LIN {X 0,Y 476.496,Z 164.694,A -85,B 0,C 180,E1 -7312.32,E2 -7312.32} C_VEL
LIN {X 0,Y 474.632,Z 154.455,A -85,B 0,C 180,E1 -7314.435,E2 -7314.435} C_VEL
LIN {X 0,Y 474.635,Z 154.349,A -85,B 0,C 180,E1 -7317.323,E2 -7317.323} C_VEL
LIN {X 0,Y 474.598,Z 154.362,A -85,B 0,C 180,E1 -7320.229,E2 -7320.229} C_VEL
LIN {X 0,Y 474.631,Z 154.36,A -85,B 0,C 180,E1 -7323.22,E2 -7323.22} C_VEL
LIN {X 0,Y 474.579,Z 154.367,A -85,B 0,C 180,E1 -7326.323,E2 -7326.323} C_VEL
LIN {X 0,Y 474.62,Z 154.363,A -85,B 0,C 180,E1 -7329.547,E2 -7329.547} C_VEL
LIN {X 0,Y 474.593,Z 154.363,A -85,B 0,C 180,E1 -7332.232,E2 -7332.232} C_VEL
LIN {X 0,Y 474.614,Z 154.365,A -85,B 0,C 180,E1 -7335.296,E2 -7335.296} C_VEL
LIN {X 0,Y 474.612,Z 154.36,A -85,B 0,C 180,E1 -7338.214,E2 -7338.214} C_VEL
LIN {X 0,Y 474.602,Z 154.355,A -85,B 0,C 180,E1 -7341.542,E2 -7341.542} C_VEL
LIN {X 0,Y 474.614,Z 154.352,A -85,B 0,C 180,E1 -7344.725,E2 -7344.725} C_VEL
LIN {X 0,Y 474.624,Z 154.36,A -85,B 0,C 180,E1 -7347.787,E2 -7347.787} C_VEL
LIN {X 0,Y 474.611,Z 154.363,A -85,B 0,C 180,E1 -7350.884,E2 -7350.884} C_VEL
LIN {X 0,Y 474.642,Z 154.358,A -85,B 0,C 180,E1 -7353.627,E2 -7353.627} C_VEL
LIN {X 0,Y 474.623,Z 154.359,A -85,B 0,C 180,E1 -7356.641,E2 -7356.641} C_VEL
LIN {X 0,Y 474.642,Z 154.358,A -85,B 0,C 180,E1 -7360.089,E2 -7360.089} C_VEL
LIN {X 0,Y 474.626,Z 154.36,A -85,B 0,C 180,E1 -7362.774,E2 -7362.774} C_VEL
LIN {X 0,Y 474.634,Z 154.359,A -85,B 0,C 180,E1 -7365.421,E2 -7365.421} C_VEL
LIN {X 0,Y 474.728,Z 154.343,A -85,B 0,C 180,E1 -7368.038,E2 -7368.038} C_VEL
LIN {X 0,Y 474.714,Z 154.348,A -85,B 0,C 180,E1 -7371.486,E2 -7371.486} C_VEL
LIN {X 0,Y 474.756,Z 154.343,A -85,B 0,C 180,E1 -7374.052,E2 -7374.052} C_VEL
LIN {X 0,Y 474.879,Z 154.327,A -85,B 0,C 180,E1 -7377.455,E2 -7377.455} C_VEL
LIN {X 0,Y 474.844,Z 154.331,A -85,B 0,C 180,E1 -7380.848,E2 -7380.848} C_VEL
LIN {X 0,Y 474.879,Z 154.327,A -85,B 0,C 180,E1 -7382.545,E2 -7382.545} C_VEL
LIN {X 0,Y 474.756,Z 154.345,A -85,B 0,C 180,E1 -7385.948,E2 -7385.948} C_VEL
LIN {X 0,Y 474.715,Z 154.346,A -85,B 0,C 180,E1 -7388.514,E2 -7388.514} C_VEL
LIN {X 0,Y 474.692,Z 154.353,A -85,B 0,C 180,E1 -7391.963,E2 -7391.963} C_VEL
LIN {X 0,Y 474.687,Z 154.346,A -85,B 0,C 180,E1 -7395.456,E2 -7395.456} C_VEL
LIN {X 0,Y 474.654,Z 154.356,A -85,B 0,C 180,E1 -7399.011,E2 -7399.011} C_VEL
LIN {X 0,Y 474.582,Z 154.363,A -85,B 0,C 180,E1 -7401.729,E2 -7401.729} C_VEL
LIN {X 0,Y 474.648,Z 154.361,A -85,B 0,C 180,E1 -7404.494,E2 -7404.494} C_VEL
LIN {X 0,Y 474.671,Z 154.35,A -85,B 0,C 180,E1 -7407.335,E2 -7407.335} C_VEL
LIN {X 0,Y 474.595,Z 154.37,A -85,B 0,C 180,E1 -7410.231,E2 -7410.231} C_VEL
LIN {X 0,Y 474.633,Z 154.352,A -85,B 0,C 180,E1 -7413.221,E2 -7413.221} C_VEL
LIN {X 0,Y 474.583,Z 154.357,A -85,B 0,C 180,E1 -7416.324,E2 -7416.324} C_VEL
LIN {X 0,Y 474.619,Z 154.364,A -85,B 0,C 180,E1 -7419.649,E2 -7419.649} C_VEL
LIN {X 0,Y 474.599,Z 154.351,A -85,B 0,C 180,E1 -7422.936,E2 -7422.936} C_VEL
LIN {X 0,Y 474.598,Z 154.367,A -85,B 0,C 180,E1 -7425.896,E2 -7425.896} C_VEL
LIN {X 0,Y 474.622,Z 154.355,A -85,B 0,C 180,E1 -7429.042,E2 -7429.042} C_VEL
LIN {X 0,Y 474.605,Z 154.362,A -85,B 0,C 180,E1 -7431.705,E2 -7431.705} C_VEL
LIN {X 0,Y 474.624,Z 154.355,A -85,B 0,C 180,E1 -7434.727,E2 -7434.727} C_VEL
LIN {X 0,Y 474.633,Z 154.363,A -85,B 0,C 180,E1 -7437.789,E2 -7437.789} C_VEL
LIN {X 0,Y 474.621,Z 154.362,A -85,B 0,C 180,E1 -7440.886,E2 -7440.886} C_VEL
LIN {X 0,Y 474.657,Z 154.36,A -85,B 0,C 180,E1 -7443.629,E2 -7443.629} C_VEL
LIN {X 0,Y 474.661,Z 154.46,A -85,B 0,C 180,E1 -7446.902,E2 -7446.902} C_VEL
LIN {X 0,Y 476.247,Z 163.612,A -85,B 0,C 180,E1 -7448.865,E2 -7448.865} C_VEL
LIN {X 0,Y 476.003,Z 169.231,A -85,B 0,C 180,E1 -7449.97,E2 -7449.97} C_VEL
LIN {X 0,Y 475.26,Z 171.385,A -85,B 0,C 180,E1 -7450.363,E2 -7450.363} C_VEL
LIN {X 0,Y 472.299,Z 175.015,A -85,B 0,C 180,E1 -7450.95,E2 -7450.95} C_VEL
LIN {X 0,Y 469.331,Z 178.656,A -85,B 0,C 180,E1 -7451.543,E2 -7451.543} C_VEL
LIN {X 0,Y 468.592,Z 180.83,A -85,B 0,C 180,E1 -7451.942,E2 -7451.942} C_VEL
LIN {X 0,Y 468.452,Z 186.605,A -85,B 0,C 180,E1 -7453.017,E2 -7453.017} C_VEL
LIN {X 0,Y 471.25,Z 202.144,A -85,B 0,C 180,E1 -7453.391,E2 -7453.391} C_VEL
LIN {X 0,Y 470.685,Z 294.202,A -85,B 0,C 180,E1 -7454.826,E2 -7454.826} C_VEL
LIN {X 0,Y 470.344,Z 307.324,A -85,B 0,C 180,E1 -7455.202,E2 -7455.202} C_VEL
LIN {X 0,Y 469.901,Z 319.4,A -85,B 0,C 180,E1 -7455.714,E2 -7455.714} C_VEL
LIN {X 0,Y 469.477,Z 330.795,A -85,B 0,C 180,E1 -7456.364,E2 -7456.364} C_VEL
LIN {X 0,Y 469.045,Z 342.481,A -85,B 0,C 180,E1 -7457.232,E2 -7457.232} C_VEL
LIN {X 0,Y 468.521,Z 352.971,A -85,B 0,C 180,E1 -7458.207,E2 -7458.207} C_VEL
LIN {X 0,Y 468.048,Z 361.544,A -85,B 0,C 180,E1 -7459.182,E2 -7459.182} C_VEL
LIN {X 0,Y 467.675,Z 369.442,A -85,B 0,C 180,E1 -7460.267,E2 -7460.267} C_VEL
LIN {X 0,Y 467.268,Z 377.166,A -85,B 0,C 180,E1 -7461.568,E2 -7461.568} C_VEL
LIN {X 0,Y 466.994,Z 384.254,A -85,B 0,C 180,E1 -7463.086,E2 -7463.086} C_VEL
LIN {X 0,Y 466.881,Z 388.978,A -85,B 0,C 180,E1 -7464.385,E2 -7464.385} C_VEL
LIN {X 0,Y 466.691,Z 392.597,A -85,B 0,C 180,E1 -7465.682,E2 -7465.682} C_VEL
LIN {X 0,Y 466.746,Z 394.466,A -85,B 0,C 180,E1 -7466.547,E2 -7466.547} C_VEL
LIN {X 0,Y 466.669,Z 395.877,A -85,B 0,C 180,E1 -7467.411,E2 -7467.411} C_VEL
LIN {X 0,Y 466.59,Z 397.498,A -85,B 0,C 180,E1 -7469.137,E2 -7469.137} C_VEL
LIN {X 0,Y 466.599,Z 397.734,A -85,B 0,C 180,E1 -7470,E2 -7470} C_VEL
LIN {X 0,Y 466.59,Z 397.547,A -85,B 0,C 180,E1 -7470.863,E2 -7470.863} C_VEL
LIN {X 0,Y 466.669,Z 395.992,A -85,B 0,C 180,E1 -7472.59,E2 -7472.59} C_VEL
LIN {X 0,Y 466.745,Z 394.631,A -85,B 0,C 180,E1 -7473.453,E2 -7473.453} C_VEL
LIN {X 0,Y 466.712,Z 391.756,A -85,B 0,C 180,E1 -7474.751,E2 -7474.751} C_VEL
LIN {X 0,Y 466.89,Z 387.046,A -85,B 0,C 180,E1 -7476.28,E2 -7476.28} C_VEL
LIN {X 0,Y 467.102,Z 380.85,A -85,B 0,C 180,E1 -7477.783,E2 -7477.783} C_VEL
LIN {X 0,Y 467.471,Z 374.044,A -85,B 0,C 180,E1 -7479.083,E2 -7479.083} C_VEL
LIN {X 0,Y 467.839,Z 365.548,A -85,B 0,C 180,E1 -7480.385,E2 -7480.385} C_VEL
LIN {X 0,Y 468.279,Z 356.811,A -85,B 0,C 180,E1 -7481.47,E2 -7481.47} C_VEL
LIN {X 0,Y 468.838,Z 346.297,A -85,B 0,C 180,E1 -7482.531,E2 -7482.531} C_VEL
LIN {X 0,Y 469.248,Z 335.279,A -85,B 0,C 180,E1 -7483.423,E2 -7483.423} C_VEL
LIN {X 0,Y 469.803,Z 323.169,A -85,B 0,C 180,E1 -7484.18,E2 -7484.18} C_VEL
LIN {X 0,Y 470.239,Z 310.502,A -85,B 0,C 180,E1 -7484.774,E2 -7484.774} C_VEL
LIN {X 0,Y 470.602,Z 297.977,A -85,B 0,C 180,E1 -7485.178,E2 -7485.178} C_VEL
LIN {X 0,Y 470.757,Z 281.99,A -85,B 0,C 180,E1 -7485.477,E2 -7485.477} C_VEL
LIN {X 0,Y 471.183,Z 201.775,A -85,B 0,C 180,E1 -7486.71,E2 -7486.71} C_VEL
LIN {X 0,Y 468.503,Z 186.823,A -85,B 0,C 180,E1 -7487.063,E2 -7487.063} C_VEL
LIN {X 0,Y 468.44,Z 185.986,A -85,B 0,C 180,E1 -7487.157,E2 -7487.157} C_VEL
LIN {X 0,Y 469.081,Z 169.504,A -85,B 0,C 180,E1 -7490.386,E2 -7490.386} C_VEL
LIN {X 0,Y 469.266,Z 164.503,A -85,B 0,C 180,E1 -7491.386,E2 -7491.386} C_VEL
LIN {X 0,Y 467.613,Z 155.303,A -85,B 0,C 180,E1 -7493.404,E2 -7493.404} C_VEL
LIN {X 0,Y 467.618,Z 155.238,A -85,B 0,C 180,E1 -7496.8,E2 -7496.8} C_VEL
LIN {X 0,Y 467.555,Z 155.243,A -85,B 0,C 180,E1 -7499.738,E2 -7499.738} C_VEL
LIN {X 0,Y 467.584,Z 155.241,A -85,B 0,C 180,E1 -7502.758,E2 -7502.758} C_VEL
LIN {X 0,Y 467.556,Z 155.238,A -85,B 0,C 180,E1 -7505.889,E2 -7505.889} C_VEL
LIN {X 0,Y 467.559,Z 155.234,A -85,B 0,C 180,E1 -7509.146,E2 -7509.146} C_VEL
LIN {X 0,Y 467.585,Z 155.24,A -85,B 0,C 180,E1 -7512.566,E2 -7512.566} C_VEL
LIN {X 0,Y 467.563,Z 155.235,A -85,B 0,C 180,E1 -7515.052,E2 -7515.052} C_VEL
LIN {X 0,Y 467.587,Z 155.225,A -85,B 0,C 180,E1 -7517.439,E2 -7517.439} C_VEL
LIN {X 0,Y 467.579,Z 155.238,A -85,B 0,C 180,E1 -7520.855,E2 -7520.855} C_VEL
LIN {X 0,Y 467.558,Z 155.223,A -85,B 0,C 180,E1 -7524.26,E2 -7524.26} C_VEL
LIN {X 0,Y 467.577,Z 155.232,A -85,B 0,C 180,E1 -7527.32,E2 -7527.32} C_VEL
LIN {X 0,Y 467.565,Z 155.239,A -85,B 0,C 180,E1 -7530.667,E2 -7530.667} C_VEL
LIN {X 0,Y 467.607,Z 155.23,A -85,B 0,C 180,E1 -7533.199,E2 -7533.199} C_VEL
LIN {X 0,Y 467.584,Z 155.235,A -85,B 0,C 180,E1 -7536.469,E2 -7536.469} C_VEL
LIN {X 0,Y 467.616,Z 155.237,A -85,B 0,C 180,E1 -7539.777,E2 -7539.777} C_VEL
LIN {X 0,Y 467.6,Z 155.233,A -85,B 0,C 180,E1 -7542.506,E2 -7542.506} C_VEL
LIN {X 0,Y 467.599,Z 155.23,A -85,B 0,C 180,E1 -7545.196,E2 -7545.196} C_VEL
LIN {X 0,Y 467.649,Z 155.233,A -85,B 0,C 180,E1 -7547.854,E2 -7547.854} C_VEL
LIN {X 0,Y 467.674,Z 155.221,A -85,B 0,C 180,E1 -7551.357,E2 -7551.357} C_VEL
LIN {X 0,Y 467.726,Z 155.222,A -85,B 0,C 180,E1 -7553.962,E2 -7553.962} C_VEL
LIN {X 0,Y 467.849,Z 155.202,A -85,B 0,C 180,E1 -7557.417,E2 -7557.417} C_VEL
LIN {X 0,Y 467.872,Z 155.203,A -85,B 0,C 180,E1 -7560,E2 -7560} C_VEL
LIN {X 0,Y 467.85,Z 155.202,A -85,B 0,C 180,E1 -7562.583,E2 -7562.583} C_VEL
LIN {X 0,Y 467.725,Z 155.218,A -85,B 0,C 180,E1 -7566.038,E2 -7566.038} C_VEL
LIN {X 0,Y 467.662,Z 155.227,A -85,B 0,C 180,E1 -7568.643,E2 -7568.643} C_VEL
LIN {X 0,Y 467.648,Z 155.225,A -85,B 0,C 180,E1 -7572.146,E2 -7572.146} C_VEL
LIN {X 0,Y 467.632,Z 155.232,A -85,B 0,C 180,E1 -7575.695,E2 -7575.695} C_VEL
LIN {X 0,Y 467.615,Z 155.236,A -85,B 0,C 180,E1 -7579.308,E2 -7579.308} C_VEL
LIN {X 0,Y 467.527,Z 155.243,A -85,B 0,C 180,E1 -7582.074,E2 -7582.074} C_VEL
LIN {X 0,Y 467.578,Z 155.236,A -85,B 0,C 180,E1 -7584.889,E2 -7584.889} C_VEL
LIN {X 0,Y 467.613,Z 155.233,A -85,B 0,C 180,E1 -7587.77,E2 -7587.77} C_VEL
LIN {X 0,Y 467.562,Z 155.244,A -85,B 0,C 180,E1 -7591.045,E2 -7591.045} C_VEL
LIN {X 0,Y 467.572,Z 155.235,A -85,B 0,C 180,E1 -7594.241,E2 -7594.241} C_VEL
LIN {X 0,Y 467.543,Z 155.231,A -85,B 0,C 180,E1 -7597.187,E2 -7597.187} C_VEL
LIN {X 0,Y 467.567,Z 155.239,A -85,B 0,C 180,E1 -7600.266,E2 -7600.266} C_VEL
LIN {X 0,Y 467.545,Z 155.241,A -85,B 0,C 180,E1 -7603.746,E2 -7603.746} C_VEL
LIN {X 0,Y 467.544,Z 155.243,A -85,B 0,C 180,E1 -7606.255,E2 -7606.255} C_VEL
LIN {X 0,Y 467.557,Z 155.239,A -85,B 0,C 180,E1 -7609.734,E2 -7609.734} C_VEL
LIN {X 0,Y 467.541,Z 155.242,A -85,B 0,C 180,E1 -7612.815,E2 -7612.815} C_VEL
LIN {X 0,Y 467.583,Z 155.234,A -85,B 0,C 180,E1 -7616.212,E2 -7616.212} C_VEL
LIN {X 0,Y 467.567,Z 155.238,A -85,B 0,C 180,E1 -7619.266,E2 -7619.266} C_VEL
LIN {X 0,Y 467.604,Z 155.225,A -85,B 0,C 180,E1 -7622.469,E2 -7622.469} C_VEL
LIN {X 0,Y 467.608,Z 155.32,A -85,B 0,C 180,E1 -7625.35,E2 -7625.35} C_VEL
LIN {X 0,Y 469.554,Z 165.837,A -85,B 0,C 180,E1 -7627.563,E2 -7627.563} C_VEL
LIN {X 0,Y 469.08,Z 177.76,A -85,B 0,C 180,E1 -7629.843,E2 -7629.843} C_VEL
LIN {X 0,Y 468.446,Z 192.056,A -85,B 0,C 180,E1 -7632.539,E2 -7632.539} C_VEL
LIN {X 0,Y 468.409,Z 194.559,A -85,B 0,C 180,E1 -7632.963,E2 -7632.963} C_VEL
LIN {X 0,Y 471.306,Z 212.054,A -85,B 0,C 180,E1 -7633.371,E2 -7633.371} C_VEL
LIN {X 0,Y 470.62,Z 302.152,A -85,B 0,C 180,E1 -7634.768,E2 -7634.768} C_VEL
LIN {X 0,Y 470.222,Z 315.409,A -85,B 0,C 180,E1 -7635.142,E2 -7635.142} C_VEL
LIN {X 0,Y 469.849,Z 327.558,A -85,B 0,C 180,E1 -7635.656,E2 -7635.656} C_VEL
LIN {X 0,Y 469.374,Z 339.815,A -85,B 0,C 180,E1 -7636.36,E2 -7636.36} C_VEL
LIN {X 0,Y 468.891,Z 350.559,A -85,B 0,C 180,E1 -7637.157,E2 -7637.157} C_VEL
LIN {X 0,Y 468.41,Z 361.811,A -85,B 0,C 180,E1 -7638.204,E2 -7638.204} C_VEL
LIN {X 0,Y 467.898,Z 370.327,A -85,B 0,C 180,E1 -7639.178,E2 -7639.178} C_VEL
LIN {X 0,Y 467.514,Z 378.184,A -85,B 0,C 180,E1 -7640.263,E2 -7640.263} C_VEL
LIN {X 0,Y 467.179,Z 385.855,A -85,B 0,C 180,E1 -7641.566,E2 -7641.566} C_VEL
LIN {X 0,Y 466.855,Z 392.925,A -85,B 0,C 180,E1 -7643.083,E2 -7643.083} C_VEL
LIN {X 0,Y 466.801,Z 397.628,A -85,B 0,C 180,E1 -7644.384,E2 -7644.384} C_VEL
LIN {X 0,Y 466.648,Z 401.219,A -85,B 0,C 180,E1 -7645.681,E2 -7645.681} C_VEL
LIN {X 0,Y 466.69,Z 403.072,A -85,B 0,C 180,E1 -7646.546,E2 -7646.546} C_VEL
LIN {X 0,Y 466.646,Z 404.461,A -85,B 0,C 180,E1 -7647.41,E2 -7647.41} C_VEL
LIN {X 0,Y 466.589,Z 406.056,A -85,B 0,C 180,E1 -7649.137,E2 -7649.137} C_VEL
LIN {X 0,Y 466.598,Z 406.272,A -85,B 0,C 180,E1 -7650,E2 -7650} C_VEL
LIN {X 0,Y 466.604,Z 405.452,A -85,B 0,C 180,E1 -7651.726,E2 -7651.726} C_VEL
LIN {X 0,Y 466.646,Z 404.463,A -85,B 0,C 180,E1 -7652.589,E2 -7652.589} C_VEL
LIN {X 0,Y 466.689,Z 403.074,A -85,B 0,C 180,E1 -7653.453,E2 -7653.453} C_VEL
LIN {X 0,Y 466.692,Z 400.152,A -85,B 0,C 180,E1 -7654.751,E2 -7654.751} C_VEL
LIN {X 0,Y 466.8,Z 396.197,A -85,B 0,C 180,E1 -7656.049,E2 -7656.049} C_VEL
LIN {X 0,Y 466.988,Z 390.112,A -85,B 0,C 180,E1 -7657.566,E2 -7657.566} C_VEL
LIN {X 0,Y 467.303,Z 383.46,A -85,B 0,C 180,E1 -7658.867,E2 -7658.867} C_VEL
LIN {X 0,Y 467.693,Z 375.204,A -85,B 0,C 180,E1 -7660.169,E2 -7660.169} C_VEL
LIN {X 0,Y 468.102,Z 366.74,A -85,B 0,C 180,E1 -7661.255,E2 -7661.255} C_VEL
LIN {X 0,Y 468.662,Z 356.491,A -85,B 0,C 180,E1 -7662.318,E2 -7662.318} C_VEL
LIN {X 0,Y 469.058,Z 346.211,A -85,B 0,C 180,E1 -7663.185,E2 -7663.185} C_VEL
LIN {X 0,Y 469.515,Z 334.567,A -85,B 0,C 180,E1 -7663.967,E2 -7663.967} C_VEL
LIN {X 0,Y 469.994,Z 322.917,A -85,B 0,C 180,E1 -7664.56,E2 -7664.56} C_VEL
LIN {X 0,Y 470.42,Z 309.487,A -85,B 0,C 180,E1 -7665.044,E2 -7665.044} C_VEL
LIN {X 0,Y 470.693,Z 296.212,A -85,B 0,C 180,E1 -7665.34,E2 -7665.34} C_VEL
LIN {X 0,Y 471.296,Z 211.905,A -85,B 0,C 180,E1 -7666.629,E2 -7666.629} C_VEL
LIN {X 0,Y 468.42,Z 194.62,A -85,B 0,C 180,E1 -7667.029,E2 -7667.029} C_VEL
LIN {X 0,Y 468.91,Z 181.321,A -85,B 0,C 180,E1 -7669.479,E2 -7669.479} C_VEL
LIN {X 0,Y 469.584,Z 167.014,A -85,B 0,C 180,E1 -7672.203,E2 -7672.203} C_VEL
LIN {X 0,Y 468.738,Z 161.245,A -85,B 0,C 180,E1 -7673.37,E2 -7673.37} C_VEL
LIN {X 0,Y 467.606,Z 155.311,A -85,B 0,C 180,E1 -7674.649,E2 -7674.649} C_VEL
LIN {X 0,Y 467.578,Z 155.231,A -85,B 0,C 180,E1 -7677.771,E2 -7677.771} C_VEL
LIN {X 0,Y 467.564,Z 155.24,A -85,B 0,C 180,E1 -7681.044,E2 -7681.044} C_VEL
LIN {X 0,Y 467.584,Z 155.233,A -85,B 0,C 180,E1 -7684.241,E2 -7684.241} C_VEL
LIN {X 0,Y 467.538,Z 155.242,A -85,B 0,C 180,E1 -7687.184,E2 -7687.184} C_VEL
LIN {X 0,Y 467.564,Z 155.238,A -85,B 0,C 180,E1 -7690.264,E2 -7690.264} C_VEL
LIN {X 0,Y 467.544,Z 155.243,A -85,B 0,C 180,E1 -7693.744,E2 -7693.744} C_VEL
LIN {X 0,Y 467.549,Z 155.24,A -85,B 0,C 180,E1 -7696.255,E2 -7696.255} C_VEL
LIN {X 0,Y 467.57,Z 155.242,A -85,B 0,C 180,E1 -7698.722,E2 -7698.722} C_VEL
LIN {X 0,Y 467.556,Z 155.231,A -85,B 0,C 180,E1 -7701.954,E2 -7701.954} C_VEL
LIN {X 0,Y 467.554,Z 155.238,A -85,B 0,C 180,E1 -7705.166,E2 -7705.166} C_VEL
LIN {X 0,Y 467.571,Z 155.24,A -85,B 0,C 180,E1 -7708.259,E2 -7708.259} C_VEL
LIN {X 0,Y 467.564,Z 155.241,A -85,B 0,C 180,E1 -7711.249,E2 -7711.249} C_VEL
LIN {X 0,Y 467.585,Z 155.237,A -85,B 0,C 180,E1 -7714.159,E2 -7714.159} C_VEL
LIN {X 0,Y 467.564,Z 155.243,A -85,B 0,C 180,E1 -7716.995,E2 -7716.995} C_VEL
LIN {X 0,Y 467.61,Z 155.233,A -85,B 0,C 180,E1 -7719.777,E2 -7719.777} C_VEL
LIN {X 0,Y 467.586,Z 155.234,A -85,B 0,C 180,E1 -7722.506,E2 -7722.506} C_VEL
LIN {X 0,Y 467.592,Z 155.238,A -85,B 0,C 180,E1 -7725.196,E2 -7725.196} C_VEL
LIN {X 0,Y 467.671,Z 155.221,A -85,B 0,C 180,E1 -7727.855,E2 -7727.855} C_VEL
LIN {X 0,Y 467.668,Z 155.227,A -85,B 0,C 180,E1 -7731.357,E2 -7731.357} C_VEL
LIN {X 0,Y 467.72,Z 155.218,A -85,B 0,C 180,E1 -7733.962,E2 -7733.962} C_VEL
LIN {X 0,Y 467.845,Z 155.203,A -85,B 0,C 180,E1 -7737.417,E2 -7737.417} C_VEL
LIN {X 0,Y 467.867,Z 155.203,A -85,B 0,C 180,E1 -7740,E2 -7740} C_VEL
LIN {X 0,Y 467.845,Z 155.203,A -85,B 0,C 180,E1 -7742.583,E2 -7742.583} C_VEL
LIN {X 0,Y 467.721,Z 155.222,A -85,B 0,C 180,E1 -7746.038,E2 -7746.038} C_VEL
LIN {X 0,Y 467.669,Z 155.222,A -85,B 0,C 180,E1 -7748.643,E2 -7748.643} C_VEL
LIN {X 0,Y 467.643,Z 155.233,A -85,B 0,C 180,E1 -7752.146,E2 -7752.146} C_VEL
LIN {X 0,Y 467.627,Z 155.226,A -85,B 0,C 180,E1 -7755.696,E2 -7755.696} C_VEL
LIN {X 0,Y 467.606,Z 155.236,A -85,B 0,C 180,E1 -7758.765,E2 -7758.765} C_VEL
LIN {X 0,Y 467.571,Z 155.234,A -85,B 0,C 180,E1 -7761.269,E2 -7761.269} C_VEL
LIN {X 0,Y 467.563,Z 155.241,A -85,B 0,C 180,E1 -7763.944,E2 -7763.944} C_VEL
LIN {X 0,Y 467.606,Z 155.231,A -85,B 0,C 180,E1 -7766.801,E2 -7766.801} C_VEL
LIN {X 0,Y 467.544,Z 155.243,A -85,B 0,C 180,E1 -7769.739,E2 -7769.739} C_VEL
LIN {X 0,Y 467.574,Z 155.232,A -85,B 0,C 180,E1 -7772.759,E2 -7772.759} C_VEL
LIN {X 0,Y 467.547,Z 155.226,A -85,B 0,C 180,E1 -7775.89,E2 -7775.89} C_VEL
LIN {X 0,Y 467.574,Z 155.238,A -85,B 0,C 180,E1 -7779.146,E2 -7779.146} C_VEL
LIN {X 0,Y 467.58,Z 155.227,A -85,B 0,C 180,E1 -7782.568,E2 -7782.568} C_VEL
LIN {X 0,Y 467.559,Z 155.235,A -85,B 0,C 180,E1 -7785.054,E2 -7785.054} C_VEL
LIN {X 0,Y 467.583,Z 155.24,A -85,B 0,C 180,E1 -7787.441,E2 -7787.441} C_VEL
LIN {X 0,Y 467.555,Z 155.234,A -85,B 0,C 180,E1 -7790.854,E2 -7790.854} C_VEL
LIN {X 0,Y 467.558,Z 155.237,A -85,B 0,C 180,E1 -7794.262,E2 -7794.262} C_VEL
LIN {X 0,Y 467.579,Z 155.241,A -85,B 0,C 180,E1 -7797.322,E2 -7797.322} C_VEL
LIN {X 0,Y 467.567,Z 155.241,A -85,B 0,C 180,E1 -7800.669,E2 -7800.669} C_VEL
LIN {X 0,Y 467.614,Z 155.238,A -85,B 0,C 180,E1 -7803.201,E2 -7803.201} C_VEL
LIN {X 0,Y 467.618,Z 155.252,A -85,B 0,C 180,E1 -7806.627,E2 -7806.627} C_VEL
LIN {X 0,Y 467.7,Z 155.798,A -85,B 0,C 180,E1 -7806.847,E2 -7806.847} C_VEL
LIN {X 0,Y 469.198,Z 164.087,A -85,B 0,C 180,E1 -7808.62,E2 -7808.62} C_VEL
LIN {X 0,Y 468.839,Z 175.747,A -85,B 0,C 180,E1 -7810.945,E2 -7810.945} C_VEL
LIN {X 0,Y 468.592,Z 180.83,A -85,B 0,C 180,E1 -7811.942,E2 -7811.942} C_VEL
LIN {X 0,Y 468.359,Z 183.305,A -85,B 0,C 180,E1 -7812.302,E2 -7812.302} C_VEL
LIN {X 0,Y 467.542,Z 188.103,A -85,B 0,C 180,E1 -7812.697,E2 -7812.697} C_VEL
LIN {X 0,Y 466.477,Z 193.563,A -85,B 0,C 180,E1 -7812.946,E2 -7812.946} C_VEL
LIN {X 0,Y 465.076,Z 201.654,A -85,B 0,C 180,E1 -7813.136,E2 -7813.136} C_VEL
LIN {X 0,Y 464.452,Z 209.922,A -85,B 0,C 180,E1 -7813.262,E2 -7813.262} C_VEL
LIN {X 0,Y 463.85,Z 294.285,A -85,B 0,C 180,E1 -7814.597,E2 -7814.597} C_VEL
LIN {X 0,Y 463.475,Z 307.401,A -85,B 0,C 180,E1 -7814.978,E2 -7814.978} C_VEL
LIN {X 0,Y 463.005,Z 320.582,A -85,B 0,C 180,E1 -7815.552,E2 -7815.552} C_VEL
LIN {X 0,Y 462.51,Z 332.459,A -85,B 0,C 180,E1 -7816.266,E2 -7816.266} C_VEL
LIN {X 0,Y 462.058,Z 343.922,A -85,B 0,C 180,E1 -7817.155,E2 -7817.155} C_VEL
LIN {X 0,Y 461.512,Z 354.103,A -85,B 0,C 180,E1 -7818.137,E2 -7818.137} C_VEL
LIN {X 0,Y 460.983,Z 363.314,A -85,B 0,C 180,E1 -7819.237,E2 -7819.237} C_VEL
LIN {X 0,Y 460.49,Z 372.258,A -85,B 0,C 180,E1 -7820.558,E2 -7820.558} C_VEL
LIN {X 0,Y 460.107,Z 379.461,A -85,B 0,C 180,E1 -7821.878,E2 -7821.878} C_VEL
LIN {X 0,Y 459.895,Z 385.855,A -85,B 0,C 180,E1 -7823.373,E2 -7823.373} C_VEL
LIN {X 0,Y 459.738,Z 390.365,A -85,B 0,C 180,E1 -7824.738,E2 -7824.738} C_VEL
LIN {X 0,Y 459.604,Z 392.663,A -85,B 0,C 180,E1 -7825.616,E2 -7825.616} C_VEL
LIN {X 0,Y 459.643,Z 394.532,A -85,B 0,C 180,E1 -7826.494,E2 -7826.494} C_VEL
LIN {X 0,Y 459.593,Z 395.942,A -85,B 0,C 180,E1 -7827.371,E2 -7827.371} C_VEL
LIN {X 0,Y 459.495,Z 397.563,A -85,B 0,C 180,E1 -7829.124,E2 -7829.124} C_VEL
LIN {X 0,Y 459.501,Z 397.799,A -85,B 0,C 180,E1 -7830,E2 -7830} C_VEL
LIN {X 0,Y 459.495,Z 397.612,A -85,B 0,C 180,E1 -7830.877,E2 -7830.877} C_VEL
LIN {X 0,Y 459.593,Z 396.056,A -85,B 0,C 180,E1 -7832.63,E2 -7832.63} C_VEL
LIN {X 0,Y 459.641,Z 394.695,A -85,B 0,C 180,E1 -7833.507,E2 -7833.507} C_VEL
LIN {X 0,Y 459.643,Z 391.82,A -85,B 0,C 180,E1 -7834.824,E2 -7834.824} C_VEL
LIN {X 0,Y 459.811,Z 387.92,A -85,B 0,C 180,E1 -7836.142,E2 -7836.142} C_VEL
LIN {X 0,Y 459.97,Z 382.891,A -85,B 0,C 180,E1 -7837.462,E2 -7837.462} C_VEL
LIN {X 0,Y 460.296,Z 376.563,A -85,B 0,C 180,E1 -7838.783,E2 -7838.783} C_VEL
LIN {X 0,Y 460.681,Z 368.641,A -85,B 0,C 180,E1 -7840.104,E2 -7840.104} C_VEL
LIN {X 0,Y 461.198,Z 358.789,A -85,B 0,C 180,E1 -7841.426,E2 -7841.426} C_VEL
LIN {X 0,Y 461.783,Z 348.733,A -85,B 0,C 180,E1 -7842.499,E2 -7842.499} C_VEL
LIN {X 0,Y 462.261,Z 337.357,A -85,B 0,C 180,E1 -7843.475,E2 -7843.475} C_VEL
LIN {X 0,Y 462.736,Z 327.035,A -85,B 0,C 180,E1 -7844.176,E2 -7844.176} C_VEL
LIN {X 0,Y 463.277,Z 314.456,A -85,B 0,C 180,E1 -7844.833,E2 -7844.833} C_VEL
LIN {X 0,Y 463.644,Z 301.86,A -85,B 0,C 180,E1 -7845.298,E2 -7845.298} C_VEL
LIN {X 0,Y 463.923,Z 288.992,A -85,B 0,C 180,E1 -7845.599,E2 -7845.599} C_VEL
LIN {X 0,Y 464.467,Z 203.131,A -85,B 0,C 180,E1 -7846.938,E2 -7846.938} C_VEL
LIN {X 0,Y 461.505,Z 186.805,A -85,B 0,C 180,E1 -7847.333,E2 -7847.333} C_VEL
LIN {X 0,Y 461.603,Z 183.272,A -85,B 0,C 180,E1 -7847.957,E2 -7847.957} C_VEL
LIN {X 0,Y 462.317,Z 167.264,A -85,B 0,C 180,E1 -7851.164,E2 -7851.164} C_VEL
LIN {X 0,Y 461.596,Z 161.575,A -85,B 0,C 180,E1 -7852.373,E2 -7852.373} C_VEL
LIN {X 0,Y 460.575,Z 156.168,A -85,B 0,C 180,E1 -7853.61,E2 -7853.61} C_VEL
LIN {X 0,Y 460.565,Z 156.115,A -85,B 0,C 180,E1 -7856.265,E2 -7856.265} C_VEL
LIN {X 0,Y 460.54,Z 156.116,A -85,B 0,C 180,E1 -7859.231,E2 -7859.231} C_VEL
LIN {X 0,Y 460.532,Z 156.119,A -85,B 0,C 180,E1 -7862.284,E2 -7862.284} C_VEL
LIN {X 0,Y 460.513,Z 156.112,A -85,B 0,C 180,E1 -7865.445,E2 -7865.445} C_VEL
LIN {X 0,Y 460.533,Z 156.11,A -85,B 0,C 180,E1 -7868.895,E2 -7868.895} C_VEL
LIN {X 0,Y 460.521,Z 156.12,A -85,B 0,C 180,E1 -7872.181,E2 -7872.181} C_VEL
LIN {X 0,Y 460.51,Z 156.114,A -85,B 0,C 180,E1 -7875.41,E2 -7875.41} C_VEL
LIN {X 0,Y 460.529,Z 156.117,A -85,B 0,C 180,E1 -7878.397,E2 -7878.397} C_VEL
LIN {X 0,Y 460.523,Z 156.117,A -85,B 0,C 180,E1 -7881.266,E2 -7881.266} C_VEL
LIN {X 0,Y 460.508,Z 156.097,A -85,B 0,C 180,E1 -7884.554,E2 -7884.554} C_VEL
LIN {X 0,Y 460.527,Z 156.113,A -85,B 0,C 180,E1 -7887.715,E2 -7887.715} C_VEL
LIN {X 0,Y 460.535,Z 156.114,A -85,B 0,C 180,E1 -7890.769,E2 -7890.769} C_VEL
LIN {X 0,Y 460.55,Z 156.115,A -85,B 0,C 180,E1 -7893.734,E2 -7893.734} C_VEL
LIN {X 0,Y 460.538,Z 156.112,A -85,B 0,C 180,E1 -7896.623,E2 -7896.623} C_VEL
LIN {X 0,Y 460.544,Z 156.113,A -85,B 0,C 180,E1 -7899.452,E2 -7899.452} C_VEL
LIN {X 0,Y 460.551,Z 156.113,A -85,B 0,C 180,E1 -7902.23,E2 -7902.23} C_VEL
LIN {X 0,Y 460.558,Z 156.105,A -85,B 0,C 180,E1 -7904.965,E2 -7904.965} C_VEL
LIN {X 0,Y 460.604,Z 156.105,A -85,B 0,C 180,E1 -7908.559,E2 -7908.559} C_VEL
LIN {X 0,Y 460.688,Z 156.095,A -85,B 0,C 180,E1 -7912.108,E2 -7912.108} C_VEL
LIN {X 0,Y 460.685,Z 156.096,A -85,B 0,C 180,E1 -7914.748,E2 -7914.748} C_VEL
LIN {X 0,Y 460.79,Z 156.081,A -85,B 0,C 180,E1 -7917.377,E2 -7917.377} C_VEL
LIN {X 0,Y 460.842,Z 156.079,A -85,B 0,C 180,E1 -7920,E2 -7920} C_VEL
LIN {X 0,Y 460.791,Z 156.082,A -85,B 0,C 180,E1 -7922.623,E2 -7922.623} C_VEL
LIN {X 0,Y 460.69,Z 156.094,A -85,B 0,C 180,E1 -7926.13,E2 -7926.13} C_VEL
LIN {X 0,Y 460.612,Z 156.106,A -85,B 0,C 180,E1 -7928.776,E2 -7928.776} C_VEL
LIN {X 0,Y 460.602,Z 156.102,A -85,B 0,C 180,E1 -7932.334,E2 -7932.334} C_VEL
LIN {X 0,Y 460.594,Z 156.106,A -85,B 0,C 180,E1 -7935.998,E2 -7935.998} C_VEL
LIN {X 0,Y 460.561,Z 156.115,A -85,B 0,C 180,E1 -7939.616,E2 -7939.616} C_VEL
LIN {X 0,Y 460.504,Z 156.118,A -85,B 0,C 180,E1 -7942.429,E2 -7942.429} C_VEL
LIN {X 0,Y 460.547,Z 156.115,A -85,B 0,C 180,E1 -7945.798,E2 -7945.798} C_VEL
LIN {X 0,Y 460.546,Z 156.112,A -85,B 0,C 180,E1 -7948.234,E2 -7948.234} C_VEL
LIN {X 0,Y 460.515,Z 156.124,A -85,B 0,C 180,E1 -7951.283,E2 -7951.283} C_VEL
LIN {X 0,Y 460.518,Z 156.114,A -85,B 0,C 180,E1 -7954.504,E2 -7954.504} C_VEL
LIN {X 0,Y 460.497,Z 156.112,A -85,B 0,C 180,E1 -7957.624,E2 -7957.624} C_VEL
LIN {X 0,Y 460.531,Z 156.116,A -85,B 0,C 180,E1 -7960.269,E2 -7960.269} C_VEL
LIN {X 0,Y 460.505,Z 156.12,A -85,B 0,C 180,E1 -7963.375,E2 -7963.375} C_VEL
LIN {X 0,Y 460.5,Z 156.123,A -85,B 0,C 180,E1 -7966.625,E2 -7966.625} C_VEL
LIN {X 0,Y 460.523,Z 156.115,A -85,B 0,C 180,E1 -7969.734,E2 -7969.734} C_VEL
LIN {X 0,Y 460.495,Z 156.115,A -85,B 0,C 180,E1 -7972.525,E2 -7972.525} C_VEL
LIN {X 0,Y 460.545,Z 156.11,A -85,B 0,C 180,E1 -7975.624,E2 -7975.624} C_VEL
LIN {X 0,Y 460.537,Z 156.117,A -85,B 0,C 180,E1 -7978.745,E2 -7978.745} C_VEL
LIN {X 0,Y 460.551,Z 156.105,A -85,B 0,C 180,E1 -7982.262,E2 -7982.262} C_VEL
LIN {X 0,Y 460.577,Z 156.319,A -85,B 0,C 180,E1 -7985.189,E2 -7985.189} C_VEL
LIN {X 0,Y 462.595,Z 166.966,A -85,B 0,C 180,E1 -7987.443,E2 -7987.443} C_VEL
LIN {X 0,Y 462.122,Z 178.888,A -85,B 0,C 180,E1 -7989.758,E2 -7989.758} C_VEL
LIN {X 0,Y 461.426,Z 194.302,A -85,B 0,C 180,E1 -7992.679,E2 -7992.679} C_VEL
LIN {X 0,Y 462.153,Z 198.619,A -85,B 0,C 180,E1 -7992.819,E2 -7992.819} C_VEL
LIN {X 0,Y 464.515,Z 213.531,A -85,B 0,C 180,E1 -7993.145,E2 -7993.145} C_VEL
LIN {X 0,Y 463.788,Z 302.098,A -85,B 0,C 180,E1 -7994.538,E2 -7994.538} C_VEL
LIN {X 0,Y 463.364,Z 315.351,A -85,B 0,C 180,E1 -7994.917,E2 -7994.917} C_VEL
LIN {X 0,Y 462.984,Z 327.498,A -85,B 0,C 180,E1 -7995.439,E2 -7995.439} C_VEL
LIN {X 0,Y 462.454,Z 339.753,A -85,B 0,C 180,E1 -7996.152,E2 -7996.152} C_VEL
LIN {X 0,Y 461.933,Z 351.209,A -85,B 0,C 180,E1 -7997.021,E2 -7997.021} C_VEL
LIN {X 0,Y 461.438,Z 361.748,A -85,B 0,C 180,E1 -7998.023,E2 -7998.023} C_VEL
LIN {X 0,Y 460.907,Z 370.264,A -85,B 0,C 180,E1 -7999.012,E2 -7999.012} C_VEL
LIN {X 0,Y 460.504,Z 378.121,A -85,B 0,C 180,E1 -8000.114,E2 -8000.114} C_VEL
LIN {X 0,Y 460.135,Z 385.791,A -85,B 0,C 180,E1 -8001.436,E2 -8001.436} C_VEL
LIN {X 0,Y 459.798,Z 392.861,A -85,B 0,C 180,E1 -8002.976,E2 -8002.976} C_VEL
LIN {X 0,Y 459.72,Z 397.563,A -85,B 0,C 180,E1 -8004.297,E2 -8004.297} C_VEL
LIN {X 0,Y 459.566,Z 401.154,A -85,B 0,C 180,E1 -8005.614,E2 -8005.614} C_VEL
LIN {X 0,Y 459.585,Z 403.007,A -85,B 0,C 180,E1 -8006.493,E2 -8006.493} C_VEL
LIN {X 0,Y 459.57,Z 404.396,A -85,B 0,C 180,E1 -8007.37,E2 -8007.37} C_VEL
LIN {X 0,Y 459.494,Z 405.992,A -85,B 0,C 180,E1 -8009.123,E2 -8009.123} C_VEL
LIN {X 0,Y 459.501,Z 406.207,A -85,B 0,C 180,E1 -8010,E2 -8010} C_VEL
LIN {X 0,Y 459.516,Z 405.387,A -85,B 0,C 180,E1 -8011.752,E2 -8011.752} C_VEL
LIN {X 0,Y 459.57,Z 404.398,A -85,B 0,C 180,E1 -8012.629,E2 -8012.629} C_VEL
LIN {X 0,Y 459.584,Z 403.009,A -85,B 0,C 180,E1 -8013.506,E2 -8013.506} C_VEL
LIN {X 0,Y 459.624,Z 400.087,A -85,B 0,C 180,E1 -8014.824,E2 -8014.824} C_VEL
LIN {X 0,Y 459.723,Z 396.131,A -85,B 0,C 180,E1 -8016.143,E2 -8016.143} C_VEL
LIN {X 0,Y 459.919,Z 390.045,A -85,B 0,C 180,E1 -8017.683,E2 -8017.683} C_VEL
LIN {X 0,Y 460.248,Z 383.393,A -85,B 0,C 180,E1 -8019.004,E2 -8019.004} C_VEL
LIN {X 0,Y 460.654,Z 375.137,A -85,B 0,C 180,E1 -8020.326,E2 -8020.326} C_VEL
LIN {X 0,Y 461.123,Z 366.672,A -85,B 0,C 180,E1 -8021.427,E2 -8021.427} C_VEL
LIN {X 0,Y 461.708,Z 356.619,A -85,B 0,C 180,E1 -8022.488,E2 -8022.488} C_VEL
LIN {X 0,Y 462.126,Z 346.142,A -85,B 0,C 180,E1 -8023.387,E2 -8023.387} C_VEL
LIN {X 0,Y 462.621,Z 334.498,A -85,B 0,C 180,E1 -8024.179,E2 -8024.179} C_VEL
LIN {X 0,Y 463.115,Z 322.846,A -85,B 0,C 180,E1 -8024.781,E2 -8024.781} C_VEL
LIN {X 0,Y 463.576,Z 309.413,A -85,B 0,C 180,E1 -8025.272,E2 -8025.272} C_VEL
LIN {X 0,Y 463.867,Z 296.132,A -85,B 0,C 180,E1 -8025.572,E2 -8025.572} C_VEL
LIN {X 0,Y 464.389,Z 211.821,A -85,B 0,C 180,E1 -8026.883,E2 -8026.883} C_VEL
LIN {X 0,Y 461.451,Z 194.534,A -85,B 0,C 180,E1 -8027.296,E2 -8027.296} C_VEL
LIN {X 0,Y 461.808,Z 185.303,A -85,B 0,C 180,E1 -8029.006,E2 -8029.006} C_VEL
LIN {X 0,Y 462.632,Z 168.14,A -85,B 0,C 180,E1 -8032.319,E2 -8032.319} C_VEL
LIN {X 0,Y 461.363,Z 160.318,A -85,B 0,C 180,E1 -8033.937,E2 -8033.937} C_VEL
LIN {X 0,Y 460.537,Z 156.17,A -85,B 0,C 180,E1 -8034.872,E2 -8034.872} C_VEL
LIN {X 0,Y 460.524,Z 156.116,A -85,B 0,C 180,E1 -8038.234,E2 -8038.234} C_VEL
LIN {X 0,Y 460.517,Z 156.121,A -85,B 0,C 180,E1 -8041.282,E2 -8041.282} C_VEL
LIN {X 0,Y 460.527,Z 156.113,A -85,B 0,C 180,E1 -8044.504,E2 -8044.504} C_VEL
LIN {X 0,Y 460.493,Z 156.113,A -85,B 0,C 180,E1 -8047.622,E2 -8047.622} C_VEL
LIN {X 0,Y 460.521,Z 156.122,A -85,B 0,C 180,E1 -8051.011,E2 -8051.011} C_VEL
LIN {X 0,Y 460.509,Z 156.12,A -85,B 0,C 180,E1 -8054.588,E2 -8054.588} C_VEL
LIN {X 0,Y 460.515,Z 156.117,A -85,B 0,C 180,E1 -8057.818,E2 -8057.818} C_VEL
LIN {X 0,Y 460.532,Z 156.112,A -85,B 0,C 180,E1 -8061.102,E2 -8061.102} C_VEL
LIN {X 0,Y 460.501,Z 156.106,A -85,B 0,C 180,E1 -8064.553,E2 -8064.553} C_VEL
LIN {X 0,Y 460.519,Z 156.118,A -85,B 0,C 180,E1 -8067.715,E2 -8067.715} C_VEL
LIN {X 0,Y 460.527,Z 156.116,A -85,B 0,C 180,E1 -8070.768,E2 -8070.768} C_VEL
LIN {X 0,Y 460.545,Z 156.114,A -85,B 0,C 180,E1 -8073.734,E2 -8073.734} C_VEL
LIN {X 0,Y 460.532,Z 156.114,A -85,B 0,C 180,E1 -8076.623,E2 -8076.623} C_VEL
LIN {X 0,Y 460.539,Z 156.115,A -85,B 0,C 180,E1 -8079.452,E2 -8079.452} C_VEL
LIN {X 0,Y 460.537,Z 156.11,A -85,B 0,C 180,E1 -8082.229,E2 -8082.229} C_VEL
LIN {X 0,Y 460.552,Z 156.117,A -85,B 0,C 180,E1 -8084.964,E2 -8084.964} C_VEL
LIN {X 0,Y 460.617,Z 156.1,A -85,B 0,C 180,E1 -8087.666,E2 -8087.666} C_VEL
LIN {X 0,Y 460.616,Z 156.106,A -85,B 0,C 180,E1 -8091.224,E2 -8091.224} C_VEL
LIN {X 0,Y 460.687,Z 156.094,A -85,B 0,C 180,E1 -8093.87,E2 -8093.87} C_VEL
LIN {X 0,Y 460.786,Z 156.082,A -85,B 0,C 180,E1 -8097.377,E2 -8097.377} C_VEL
LIN {X 0,Y 460.838,Z 156.079,A -85,B 0,C 180,E1 -8100,E2 -8100} C_VEL
LIN {X 0,Y 460.786,Z 156.081,A -85,B 0,C 180,E1 -8102.623,E2 -8102.623} C_VEL
LIN {X 0,Y 460.687,Z 156.099,A -85,B 0,C 180,E1 -8106.13,E2 -8106.13} C_VEL
LIN {X 0,Y 460.616,Z 156.099,A -85,B 0,C 180,E1 -8108.776,E2 -8108.776} C_VEL
LIN {X 0,Y 460.601,Z 156.113,A -85,B 0,C 180,E1 -8112.445,E2 -8112.445} C_VEL
LIN {X 0,Y 460.588,Z 156.105,A -85,B 0,C 180,E1 -8115.998,E2 -8115.998} C_VEL
LIN {X 0,Y 460.559,Z 156.113,A -85,B 0,C 180,E1 -8118.902,E2 -8118.902} C_VEL
LIN {X 0,Y 460.506,Z 156.115,A -85,B 0,C 180,E1 -8121.486,E2 -8121.486} C_VEL
LIN {X 0,Y 460.532,Z 156.122,A -85,B 0,C 180,E1 -8124.333,E2 -8124.333} C_VEL
LIN {X 0,Y 460.562,Z 156.107,A -85,B 0,C 180,E1 -8127.245,E2 -8127.245} C_VEL
LIN {X 0,Y 460.5,Z 156.126,A -85,B 0,C 180,E1 -8130.241,E2 -8130.241} C_VEL
LIN {X 0,Y 460.52,Z 156.11,A -85,B 0,C 180,E1 -8133.326,E2 -8133.326} C_VEL
LIN {X 0,Y 460.469,Z 156.118,A -85,B 0,C 180,E1 -8136.53,E2 -8136.53} C_VEL
LIN {X 0,Y 460.524,Z 156.122,A -85,B 0,C 180,E1 -8139.863,E2 -8139.863} C_VEL
LIN {X 0,Y 460.505,Z 156.106,A -85,B 0,C 180,E1 -8142.901,E2 -8142.901} C_VEL
LIN {X 0,Y 460.501,Z 156.121,A -85,B 0,C 180,E1 -8145.832,E2 -8145.832} C_VEL
LIN {X 0,Y 460.525,Z 156.111,A -85,B 0,C 180,E1 -8148.99,E2 -8148.99} C_VEL
LIN {X 0,Y 460.514,Z 156.112,A -85,B 0,C 180,E1 -8151.267,E2 -8151.267} C_VEL
LIN {X 0,Y 460.509,Z 156.113,A -85,B 0,C 180,E1 -8154.556,E2 -8154.556} C_VEL
LIN {X 0,Y 460.529,Z 156.121,A -85,B 0,C 180,E1 -8157.717,E2 -8157.717} C_VEL
LIN {X 0,Y 460.537,Z 156.116,A -85,B 0,C 180,E1 -8160.77,E2 -8160.77} C_VEL
LIN {X 0,Y 460.558,Z 156.115,A -85,B 0,C 180,E1 -8163.736,E2 -8163.736} C_VEL
LIN {X 0,Y 460.581,Z 156.219,A -85,B 0,C 180,E1 -8166.509,E2 -8166.509} C_VEL
LIN {X 0,Y 462.261,Z 165.67,A -85,B 0,C 180,E1 -8168.6,E2 -8168.6} C_VEL
LIN {X 0,Y 461.836,Z 177.529,A -85,B 0,C 180,E1 -8170.993,E2 -8170.993} C_VEL
LIN {X 0,Y 461.485,Z 186.504,A -85,B 0,C 180,E1 -8172.736,E2 -8172.736} C_VEL
LIN {X 0,Y 462.287,Z 191.063,A -85,B 0,C 180,E1 -8172.881,E2 -8172.881} C_VEL
LIN {X 0,Y 464.451,Z 203.926,A -85,B 0,C 180,E1 -8173.168,E2 -8173.168} C_VEL
LIN {X 0,Y 464.452,Z 209.922,A -85,B 0,C 180,E1 -8173.262,E2 -8173.262} C_VEL
LIN {X 0,Y 463.803,Z 215.769,A -85,B 0,C 180,E1 -8173.331,E2 -8173.331} C_VEL
LIN {X 0,Y 458.12,Z 234.774,A -85,B 0,C 180,E1 -8173.422,E2 -8173.422} C_VEL
LIN {X 0,Y 457.489,Z 240.62,A -85,B 0,C 180,E1 -8173.492,E2 -8173.492} C_VEL
LIN {X 0,Y 457.029,Z 294.367,A -85,B 0,C 180,E1 -8174.361,E2 -8174.361} C_VEL
LIN {X 0,Y 456.613,Z 307.477,A -85,B 0,C 180,E1 -8174.747,E2 -8174.747} C_VEL
LIN {X 0,Y 456.136,Z 320.655,A -85,B 0,C 180,E1 -8175.33,E2 -8175.33} C_VEL
LIN {X 0,Y 455.621,Z 332.53,A -85,B 0,C 180,E1 -8176.055,E2 -8176.055} C_VEL
LIN {X 0,Y 455.137,Z 343.723,A -85,B 0,C 180,E1 -8176.932,E2 -8176.932} C_VEL
LIN {X 0,Y 454.564,Z 354.172,A -85,B 0,C 180,E1 -8177.953,E2 -8177.953} C_VEL
LIN {X 0,Y 453.995,Z 363.383,A -85,B 0,C 180,E1 -8179.069,E2 -8179.069} C_VEL
LIN {X 0,Y 453.47,Z 372.326,A -85,B 0,C 180,E1 -8180.41,E2 -8180.41} C_VEL
LIN {X 0,Y 453.072,Z 379.528,A -85,B 0,C 180,E1 -8181.751,E2 -8181.751} C_VEL
LIN {X 0,Y 452.869,Z 384.388,A -85,B 0,C 180,E1 -8182.869,E2 -8182.869} C_VEL
LIN {X 0,Y 452.733,Z 389.11,A -85,B 0,C 180,E1 -8184.209,E2 -8184.209} C_VEL
LIN {X 0,Y 452.524,Z 392.729,A -85,B 0,C 180,E1 -8185.547,E2 -8185.547} C_VEL
LIN {X 0,Y 452.54,Z 394.598,A -85,B 0,C 180,E1 -8186.439,E2 -8186.439} C_VEL
LIN {X 0,Y 452.519,Z 396.008,A -85,B 0,C 180,E1 -8187.33,E2 -8187.33} C_VEL
LIN {X 0,Y 452.404,Z 397.628,A -85,B 0,C 180,E1 -8189.11,E2 -8189.11} C_VEL
LIN {X 0,Y 452.407,Z 397.864,A -85,B 0,C 180,E1 -8190,E2 -8190} C_VEL
LIN {X 0,Y 452.404,Z 397.677,A -85,B 0,C 180,E1 -8190.89,E2 -8190.89} C_VEL
LIN {X 0,Y 452.519,Z 396.12,A -85,B 0,C 180,E1 -8192.671,E2 -8192.671} C_VEL
LIN {X 0,Y 452.538,Z 394.759,A -85,B 0,C 180,E1 -8193.562,E2 -8193.562} C_VEL
LIN {X 0,Y 452.579,Z 391.884,A -85,B 0,C 180,E1 -8194.9,E2 -8194.9} C_VEL
LIN {X 0,Y 452.74,Z 387.984,A -85,B 0,C 180,E1 -8196.238,E2 -8196.238} C_VEL
LIN {X 0,Y 452.902,Z 382.954,A -85,B 0,C 180,E1 -8197.58,E2 -8197.58} C_VEL
LIN {X 0,Y 453.254,Z 376.625,A -85,B 0,C 180,E1 -8198.92,E2 -8198.92} C_VEL
LIN {X 0,Y 453.691,Z 368.703,A -85,B 0,C 180,E1 -8200.262,E2 -8200.262} C_VEL
LIN {X 0,Y 454.235,Z 358.851,A -85,B 0,C 180,E1 -8201.604,E2 -8201.604} C_VEL
LIN {X 0,Y 454.839,Z 348.958,A -85,B 0,C 180,E1 -8202.677,E2 -8202.677} C_VEL
LIN {X 0,Y 455.364,Z 337.416,A -85,B 0,C 180,E1 -8203.683,E2 -8203.683} C_VEL
LIN {X 0,Y 455.852,Z 327.093,A -85,B 0,C 180,E1 -8204.395,E2 -8204.395} C_VEL
LIN {X 0,Y 456.379,Z 315.746,A -85,B 0,C 180,E1 -8205.005,E2 -8205.005} C_VEL
LIN {X 0,Y 456.787,Z 302.826,A -85,B 0,C 180,E1 -8205.505,E2 -8205.505} C_VEL
LIN {X 0,Y 457.099,Z 289.033,A -85,B 0,C 180,E1 -8205.838,E2 -8205.838} C_VEL
LIN {X 0,Y 457.686,Z 203.967,A -85,B 0,C 180,E1 -8207.184,E2 -8207.184} C_VEL
LIN {X 0,Y 454.571,Z 186.938,A -85,B 0,C 180,E1 -8207.602,E2 -8207.602} C_VEL
LIN {X 0,Y 454.543,Z 185.51,A -85,B 0,C 180,E1 -8207.804,E2 -8207.804} C_VEL
LIN {X 0,Y 455.316,Z 169.588,A -85,B 0,C 180,E1 -8211.031,E2 -8211.031} C_VEL
LIN {X 0,Y 455.21,Z 166.164,A -85,B 0,C 180,E1 -8211.749,E2 -8211.749} C_VEL
LIN {X 0,Y 453.53,Z 157.179,A -85,B 0,C 180,E1 -8213.759,E2 -8213.759} C_VEL
LIN {X 0,Y 453.508,Z 156.994,A -85,B 0,C 180,E1 -8216.706,E2 -8216.706} C_VEL
LIN {X 0,Y 453.473,Z 156.998,A -85,B 0,C 180,E1 -8219.784,E2 -8219.784} C_VEL
LIN {X 0,Y 453.491,Z 156.994,A -85,B 0,C 180,E1 -8223.189,E2 -8223.189} C_VEL
LIN {X 0,Y 453.455,Z 157,A -85,B 0,C 180,E1 -8226.299,E2 -8226.299} C_VEL
LIN {X 0,Y 453.482,Z 156.988,A -85,B 0,C 180,E1 -8229.45,E2 -8229.45} C_VEL
LIN {X 0,Y 453.475,Z 156.993,A -85,B 0,C 180,E1 -8231.934,E2 -8231.934} C_VEL
LIN {X 0,Y 453.481,Z 156.99,A -85,B 0,C 180,E1 -8235.471,E2 -8235.471} C_VEL
LIN {X 0,Y 453.476,Z 156.991,A -85,B 0,C 180,E1 -8238.209,E2 -8238.209} C_VEL
LIN {X 0,Y 453.512,Z 156.991,A -85,B 0,C 180,E1 -8240.79,E2 -8240.79} C_VEL
LIN {X 0,Y 453.452,Z 156.983,A -85,B 0,C 180,E1 -8243.917,E2 -8243.917} C_VEL
LIN {X 0,Y 453.478,Z 156.987,A -85,B 0,C 180,E1 -8247.151,E2 -8247.151} C_VEL
LIN {X 0,Y 453.47,Z 156.997,A -85,B 0,C 180,E1 -8250.268,E2 -8250.268} C_VEL
LIN {X 0,Y 453.496,Z 156.988,A -85,B 0,C 180,E1 -8253.293,E2 -8253.293} C_VEL
LIN {X 0,Y 453.491,Z 156.993,A -85,B 0,C 180,E1 -8256.238,E2 -8256.238} C_VEL
LIN {X 0,Y 453.476,Z 156.99,A -85,B 0,C 180,E1 -8259.117,E2 -8259.117} C_VEL
LIN {X 0,Y 453.504,Z 156.994,A -85,B 0,C 180,E1 -8261.944,E2 -8261.944} C_VEL
LIN {X 0,Y 453.533,Z 156.98,A -85,B 0,C 180,E1 -8264.726,E2 -8264.726} C_VEL
LIN {X 0,Y 453.552,Z 156.984,A -85,B 0,C 180,E1 -8268.379,E2 -8268.379} C_VEL
LIN {X 0,Y 453.645,Z 156.974,A -85,B 0,C 180,E1 -8271.985,E2 -8271.985} C_VEL
LIN {X 0,Y 453.658,Z 156.971,A -85,B 0,C 180,E1 -8274.667,E2 -8274.667} C_VEL
LIN {X 0,Y 453.734,Z 156.96,A -85,B 0,C 180,E1 -8277.337,E2 -8277.337} C_VEL
LIN {X 0,Y 453.813,Z 156.954,A -85,B 0,C 180,E1 -8280,E2 -8280} C_VEL
LIN {X 0,Y 453.735,Z 156.961,A -85,B 0,C 180,E1 -8282.663,E2 -8282.663} C_VEL
LIN {X 0,Y 453.658,Z 156.97,A -85,B 0,C 180,E1 -8286.226,E2 -8286.226} C_VEL
LIN {X 0,Y 453.578,Z 156.983,A -85,B 0,C 180,E1 -8288.914,E2 -8288.914} C_VEL
LIN {X 0,Y 453.557,Z 156.979,A -85,B 0,C 180,E1 -8292.529,E2 -8292.529} C_VEL
LIN {X 0,Y 453.538,Z 156.984,A -85,B 0,C 180,E1 -8296.196,E2 -8296.196} C_VEL
LIN {X 0,Y 453.51,Z 156.988,A -85,B 0,C 180,E1 -8299.039,E2 -8299.039} C_VEL
LIN {X 0,Y 453.47,Z 156.995,A -85,B 0,C 180,E1 -8301.836,E2 -8301.836} C_VEL
LIN {X 0,Y 453.494,Z 156.988,A -85,B 0,C 180,E1 -8304.736,E2 -8304.736} C_VEL
LIN {X 0,Y 453.526,Z 156.987,A -85,B 0,C 180,E1 -8307.96,E2 -8307.96} C_VEL
LIN {X 0,Y 453.459,Z 157,A -85,B 0,C 180,E1 -8311.525,E2 -8311.525} C_VEL
LIN {X 0,Y 453.478,Z 156.99,A -85,B 0,C 180,E1 -8314.777,E2 -8314.777} C_VEL
LIN {X 0,Y 453.458,Z 156.988,A -85,B 0,C 180,E1 -8318.312,E2 -8318.312} C_VEL
LIN {X 0,Y 453.49,Z 156.995,A -85,B 0,C 180,E1 -8320.61,E2 -8320.61} C_VEL
LIN {X 0,Y 453.457,Z 156.996,A -85,B 0,C 180,E1 -8324.222,E2 -8324.222} C_VEL
LIN {X 0,Y 453.434,Z 157.002,A -85,B 0,C 180,E1 -8327.002,E2 -8327.002} C_VEL
LIN {X 0,Y 453.469,Z 156.996,A -85,B 0,C 180,E1 -8329.413,E2 -8329.413} C_VEL
LIN {X 0,Y 453.448,Z 156.997,A -85,B 0,C 180,E1 -8332.81,E2 -8332.81} C_VEL
LIN {X 0,Y 453.475,Z 156.99,A -85,B 0,C 180,E1 -8336.088,E2 -8336.088} C_VEL
LIN {X 0,Y 453.475,Z 156.993,A -85,B 0,C 180,E1 -8339.241,E2 -8339.241} C_VEL
LIN {X 0,Y 453.508,Z 156.981,A -85,B 0,C 180,E1 -8342.296,E2 -8342.296} C_VEL
LIN {X 0,Y 453.514,Z 157.038,A -85,B 0,C 180,E1 -8344.899,E2 -8344.899} C_VEL
LIN {X 0,Y 454.32,Z 161.319,A -85,B 0,C 180,E1 -8345.88,E2 -8345.88} C_VEL
LIN {X 0,Y 455.726,Z 169.46,A -85,B 0,C 180,E1 -8347.596,E2 -8347.596} C_VEL
LIN {X 0,Y 454.768,Z 188.355,A -85,B 0,C 180,E1 -8351.297,E2 -8351.297} C_VEL
LIN {X 0,Y 454.482,Z 194.215,A -85,B 0,C 180,E1 -8352.403,E2 -8352.403} C_VEL
LIN {X 0,Y 455.106,Z 198.085,A -85,B 0,C 180,E1 -8352.537,E2 -8352.537} C_VEL
LIN {X 0,Y 457.727,Z 214.229,A -85,B 0,C 180,E1 -8352.899,E2 -8352.899} C_VEL
LIN {X 0,Y 456.965,Z 302.044,A -85,B 0,C 180,E1 -8354.301,E2 -8354.301} C_VEL
LIN {X 0,Y 456.525,Z 315.294,A -85,B 0,C 180,E1 -8354.686,E2 -8354.686} C_VEL
LIN {X 0,Y 456.055,Z 328.559,A -85,B 0,C 180,E1 -8355.27,E2 -8355.27} C_VEL
LIN {X 0,Y 455.557,Z 339.689,A -85,B 0,C 180,E1 -8355.938,E2 -8355.938} C_VEL
LIN {X 0,Y 455.001,Z 350.33,A -85,B 0,C 180,E1 -8356.748,E2 -8356.748} C_VEL
LIN {X 0,Y 454.454,Z 361.685,A -85,B 0,C 180,E1 -8357.836,E2 -8357.836} C_VEL
LIN {X 0,Y 453.899,Z 370.201,A -85,B 0,C 180,E1 -8358.84,E2 -8358.84} C_VEL
LIN {X 0,Y 453.506,Z 378.058,A -85,B 0,C 180,E1 -8359.96,E2 -8359.96} C_VEL
LIN {X 0,Y 453.077,Z 385.727,A -85,B 0,C 180,E1 -8361.301,E2 -8361.301} C_VEL
LIN {X 0,Y 452.735,Z 392.797,A -85,B 0,C 180,E1 -8362.866,E2 -8362.866} C_VEL
LIN {X 0,Y 452.621,Z 397.499,A -85,B 0,C 180,E1 -8364.207,E2 -8364.207} C_VEL
LIN {X 0,Y 452.489,Z 401.09,A -85,B 0,C 180,E1 -8365.546,E2 -8365.546} C_VEL
LIN {X 0,Y 452.481,Z 402.943,A -85,B 0,C 180,E1 -8366.438,E2 -8366.438} C_VEL
LIN {X 0,Y 452.495,Z 404.332,A -85,B 0,C 180,E1 -8367.329,E2 -8367.329} C_VEL
LIN {X 0,Y 452.403,Z 405.927,A -85,B 0,C 180,E1 -8369.11,E2 -8369.11} C_VEL
LIN {X 0,Y 452.407,Z 406.142,A -85,B 0,C 180,E1 -8370,E2 -8370} C_VEL
LIN {X 0,Y 452.433,Z 405.322,A -85,B 0,C 180,E1 -8371.78,E2 -8371.78} C_VEL
LIN {X 0,Y 452.495,Z 404.332,A -85,B 0,C 180,E1 -8372.67,E2 -8372.67} C_VEL
LIN {X 0,Y 452.481,Z 402.943,A -85,B 0,C 180,E1 -8373.562,E2 -8373.562} C_VEL
LIN {X 0,Y 452.556,Z 400.021,A -85,B 0,C 180,E1 -8374.899,E2 -8374.899} C_VEL
LIN {X 0,Y 452.682,Z 395.238,A -85,B 0,C 180,E1 -8376.476,E2 -8376.476} C_VEL
LIN {X 0,Y 452.908,Z 388.97,A -85,B 0,C 180,E1 -8378.027,E2 -8378.027} C_VEL
LIN {X 0,Y 453.256,Z 382.093,A -85,B 0,C 180,E1 -8379.369,E2 -8379.369} C_VEL
LIN {X 0,Y 453.698,Z 373.487,A -85,B 0,C 180,E1 -8380.712,E2 -8380.712} C_VEL
LIN {X 0,Y 454.286,Z 364.659,A -85,B 0,C 180,E1 -8381.828,E2 -8381.828} C_VEL
LIN {X 0,Y 454.815,Z 354.947,A -85,B 0,C 180,E1 -8382.835,E2 -8382.835} C_VEL
LIN {X 0,Y 455.302,Z 344.359,A -85,B 0,C 180,E1 -8383.728,E2 -8383.728} C_VEL
LIN {X 0,Y 455.831,Z 332.508,A -85,B 0,C 180,E1 -8384.509,E2 -8384.509} C_VEL
LIN {X 0,Y 456.387,Z 320.173,A -85,B 0,C 180,E1 -8385.118,E2 -8385.118} C_VEL
LIN {X 0,Y 456.829,Z 307.51,A -85,B 0,C 180,E1 -8385.56,E2 -8385.56} C_VEL
LIN {X 0,Y 457.041,Z 294.27,A -85,B 0,C 180,E1 -8385.839,E2 -8385.839} C_VEL
LIN {X 0,Y 457.574,Z 212.435,A -85,B 0,C 180,E1 -8387.131,E2 -8387.131} C_VEL
LIN {X 0,Y 454.471,Z 194.57,A -85,B 0,C 180,E1 -8387.562,E2 -8387.562} C_VEL
LIN {X 0,Y 454.634,Z 190.72,A -85,B 0,C 180,E1 -8388.241,E2 -8388.241} C_VEL
LIN {X 0,Y 455.536,Z 172.844,A -85,B 0,C 180,E1 -8391.731,E2 -8391.731} C_VEL
LIN {X 0,Y 455.583,Z 168.072,A -85,B 0,C 180,E1 -8392.684,E2 -8392.684} C_VEL
LIN {X 0,Y 453.554,Z 157.345,A -85,B 0,C 180,E1 -8394.976,E2 -8394.976} C_VEL
LIN {X 0,Y 453.503,Z 156.996,A -85,B 0,C 180,E1 -8395.224,E2 -8395.224} C_VEL
LIN {X 0,Y 453.489,Z 156.994,A -85,B 0,C 180,E1 -8398.712,E2 -8398.712} C_VEL
LIN {X 0,Y 453.46,Z 157.001,A -85,B 0,C 180,E1 -8401.798,E2 -8401.798} C_VEL
LIN {X 0,Y 453.475,Z 156.995,A -85,B 0,C 180,E1 -8404.988,E2 -8404.988} C_VEL
LIN {X 0,Y 453.453,Z 156.987,A -85,B 0,C 180,E1 -8408.311,E2 -8408.311} C_VEL
LIN {X 0,Y 453.487,Z 156.994,A -85,B 0,C 180,E1 -8410.608,E2 -8410.608} C_VEL
LIN {X 0,Y 453.456,Z 156.997,A -85,B 0,C 180,E1 -8414.22,E2 -8414.22} C_VEL
LIN {X 0,Y 453.456,Z 156.998,A -85,B 0,C 180,E1 -8417.004,E2 -8417.004} C_VEL
LIN {X 0,Y 453.486,Z 156.996,A -85,B 0,C 180,E1 -8419.408,E2 -8419.408} C_VEL
LIN {X 0,Y 453.44,Z 156.989,A -85,B 0,C 180,E1 -8422.226,E2 -8422.226} C_VEL
LIN {X 0,Y 453.477,Z 156.991,A -85,B 0,C 180,E1 -8425.222,E2 -8425.222} C_VEL
LIN {X 0,Y 453.454,Z 157,A -85,B 0,C 180,E1 -8428.474,E2 -8428.474} C_VEL
LIN {X 0,Y 453.521,Z 156.988,A -85,B 0,C 180,E1 -8432.04,E2 -8432.04} C_VEL
LIN {X 0,Y 453.488,Z 156.989,A -85,B 0,C 180,E1 -8435.264,E2 -8435.264} C_VEL
LIN {X 0,Y 453.469,Z 156.997,A -85,B 0,C 180,E1 -8438.414,E2 -8438.414} C_VEL
LIN {X 0,Y 453.51,Z 156.987,A -85,B 0,C 180,E1 -8441.008,E2 -8441.008} C_VEL
LIN {X 0,Y 453.557,Z 156.982,A -85,B 0,C 180,E1 -8443.879,E2 -8443.879} C_VEL
LIN {X 0,Y 453.59,Z 156.975,A -85,B 0,C 180,E1 -8447.472,E2 -8447.472} C_VEL
LIN {X 0,Y 453.58,Z 156.984,A -85,B 0,C 180,E1 -8451.086,E2 -8451.086} C_VEL
LIN {X 0,Y 453.655,Z 156.97,A -85,B 0,C 180,E1 -8453.774,E2 -8453.774} C_VEL
LIN {X 0,Y 453.73,Z 156.962,A -85,B 0,C 180,E1 -8457.337,E2 -8457.337} C_VEL
LIN {X 0,Y 453.808,Z 156.954,A -85,B 0,C 180,E1 -8460,E2 -8460} C_VEL
LIN {X 0,Y 453.73,Z 156.96,A -85,B 0,C 180,E1 -8462.663,E2 -8462.663} C_VEL
LIN {X 0,Y 453.655,Z 156.976,A -85,B 0,C 180,E1 -8466.226,E2 -8466.226} C_VEL
LIN {X 0,Y 453.58,Z 156.974,A -85,B 0,C 180,E1 -8468.914,E2 -8468.914} C_VEL
LIN {X 0,Y 453.551,Z 156.989,A -85,B 0,C 180,E1 -8472.529,E2 -8472.529} C_VEL
LIN {X 0,Y 453.533,Z 156.984,A -85,B 0,C 180,E1 -8476.196,E2 -8476.196} C_VEL
LIN {X 0,Y 453.509,Z 156.991,A -85,B 0,C 180,E1 -8479.041,E2 -8479.041} C_VEL
LIN {X 0,Y 453.466,Z 156.994,A -85,B 0,C 180,E1 -8481.837,E2 -8481.837} C_VEL
LIN {X 0,Y 453.504,Z 156.993,A -85,B 0,C 180,E1 -8484.735,E2 -8484.735} C_VEL
LIN {X 0,Y 453.522,Z 156.988,A -85,B 0,C 180,E1 -8487.96,E2 -8487.96} C_VEL
LIN {X 0,Y 453.456,Z 156.998,A -85,B 0,C 180,E1 -8491.526,E2 -8491.526} C_VEL
LIN {X 0,Y 453.48,Z 156.972,A -85,B 0,C 180,E1 -8494.778,E2 -8494.778} C_VEL
LIN {X 0,Y 453.457,Z 157.001,A -85,B 0,C 180,E1 -8498.313,E2 -8498.313} C_VEL
LIN {X 0,Y 453.487,Z 156.992,A -85,B 0,C 180,E1 -8500.61,E2 -8500.61} C_VEL
LIN {X 0,Y 453.446,Z 156.986,A -85,B 0,C 180,E1 -8503.245,E2 -8503.245} C_VEL
LIN {X 0,Y 453.456,Z 156.998,A -85,B 0,C 180,E1 -8505.78,E2 -8505.78} C_VEL
LIN {X 0,Y 453.474,Z 156.993,A -85,B 0,C 180,E1 -8508.21,E2 -8508.21} C_VEL
LIN {X 0,Y 453.482,Z 156.987,A -85,B 0,C 180,E1 -8510.796,E2 -8510.796} C_VEL
LIN {X 0,Y 453.452,Z 156.998,A -85,B 0,C 180,E1 -8513.918,E2 -8513.918} C_VEL
LIN {X 0,Y 453.48,Z 156.996,A -85,B 0,C 180,E1 -8517.152,E2 -8517.152} C_VEL
LIN {X 0,Y 453.473,Z 156.999,A -85,B 0,C 180,E1 -8520.269,E2 -8520.269} C_VEL
LIN {X 0,Y 453.503,Z 156.996,A -85,B 0,C 180,E1 -8523.295,E2 -8523.295} C_VEL
LIN {X 0,Y 453.508,Z 157.1,A -85,B 0,C 180,E1 -8526.301,E2 -8526.301} C_VEL
LIN {X 0,Y 455.309,Z 166.853,A -85,B 0,C 180,E1 -8528.495,E2 -8528.495} C_VEL
LIN {X 0,Y 454.824,Z 179.429,A -85,B 0,C 180,E1 -8531.066,E2 -8531.066} C_VEL
LIN {X 0,Y 454.528,Z 186.569,A -85,B 0,C 180,E1 -8532.463,E2 -8532.463} C_VEL
LIN {X 0,Y 455.46,Z 191.66,A -85,B 0,C 180,E1 -8532.625,E2 -8532.625} C_VEL
LIN {X 0,Y 457.684,Z 204.748,A -85,B 0,C 180,E1 -8532.923,E2 -8532.923} C_VEL
LIN {X 0,Y 457.489,Z 240.62,A -85,B 0,C 180,E1 -8533.492,E2 -8533.492} C_VEL
LIN {X 0,Y 456.894,Z 246.455,A -85,B 0,C 180,E1 -8533.563,E2 -8533.563} C_VEL
LIN {X 0,Y 451.277,Z 265.45,A -85,B 0,C 180,E1 -8533.66,E2 -8533.66} C_VEL
LIN {X 0,Y 450.44,Z 271.293,A -85,B 0,C 180,E1 -8533.724,E2 -8533.724} C_VEL
LIN {X 0,Y 450.187,Z 295.588,A -85,B 0,C 180,E1 -8534.146,E2 -8534.146} C_VEL
LIN {X 0,Y 449.758,Z 308.315,A -85,B 0,C 180,E1 -8534.537,E2 -8534.537} C_VEL
LIN {X 0,Y 449.249,Z 320.729,A -85,B 0,C 180,E1 -8535.1,E2 -8535.1} C_VEL
LIN {X 0,Y 448.725,Z 332.601,A -85,B 0,C 180,E1 -8535.836,E2 -8535.836} C_VEL
LIN {X 0,Y 448.266,Z 342.447,A -85,B 0,C 180,E1 -8536.608,E2 -8536.608} C_VEL
LIN {X 0,Y 447.667,Z 353.178,A -85,B 0,C 180,E1 -8537.65,E2 -8537.65} C_VEL
LIN {X 0,Y 447.104,Z 361.75,A -85,B 0,C 180,E1 -8538.669,E2 -8538.669} C_VEL
LIN {X 0,Y 446.618,Z 369.646,A -85,B 0,C 180,E1 -8539.804,E2 -8539.804} C_VEL
LIN {X 0,Y 446.176,Z 377.368,A -85,B 0,C 180,E1 -8541.166,E2 -8541.166} C_VEL
LIN {X 0,Y 445.79,Z 384.455,A -85,B 0,C 180,E1 -8542.755,E2 -8542.755} C_VEL
LIN {X 0,Y 445.661,Z 389.177,A -85,B 0,C 180,E1 -8544.117,E2 -8544.117} C_VEL
LIN {X 0,Y 445.448,Z 392.795,A -85,B 0,C 180,E1 -8545.476,E2 -8545.476} C_VEL
LIN {X 0,Y 445.439,Z 394.664,A -85,B 0,C 180,E1 -8546.382,E2 -8546.382} C_VEL
LIN {X 0,Y 445.446,Z 396.073,A -85,B 0,C 180,E1 -8547.287,E2 -8547.287} C_VEL
LIN {X 0,Y 445.316,Z 397.693,A -85,B 0,C 180,E1 -8549.096,E2 -8549.096} C_VEL
LIN {X 0,Y 445.317,Z 397.929,A -85,B 0,C 180,E1 -8550,E2 -8550} C_VEL
LIN {X 0,Y 445.316,Z 397.741,A -85,B 0,C 180,E1 -8550.905,E2 -8550.905} C_VEL
LIN {X 0,Y 445.446,Z 396.184,A -85,B 0,C 180,E1 -8552.713,E2 -8552.713} C_VEL
LIN {X 0,Y 445.437,Z 394.824,A -85,B 0,C 180,E1 -8553.619,E2 -8553.619} C_VEL
LIN {X 0,Y 445.518,Z 391.948,A -85,B 0,C 180,E1 -8554.978,E2 -8554.978} C_VEL
LIN {X 0,Y 445.75,Z 387.045,A -85,B 0,C 180,E1 -8556.633,E2 -8556.633} C_VEL
LIN {X 0,Y 445.967,Z 381.04,A -85,B 0,C 180,E1 -8558.154,E2 -8558.154} C_VEL
LIN {X 0,Y 446.344,Z 374.233,A -85,B 0,C 180,E1 -8559.517,E2 -8559.517} C_VEL
LIN {X 0,Y 446.821,Z 365.734,A -85,B 0,C 180,E1 -8560.88,E2 -8560.88} C_VEL
LIN {X 0,Y 447.415,Z 356.995,A -85,B 0,C 180,E1 -8562.013,E2 -8562.013} C_VEL
LIN {X 0,Y 448.053,Z 346.023,A -85,B 0,C 180,E1 -8563.167,E2 -8563.167} C_VEL
LIN {X 0,Y 448.564,Z 335.449,A -85,B 0,C 180,E1 -8564.055,E2 -8564.055} C_VEL
LIN {X 0,Y 449.187,Z 323.34,A -85,B 0,C 180,E1 -8564.845,E2 -8564.845} C_VEL
LIN {X 0,Y 449.706,Z 310.666,A -85,B 0,C 180,E1 -8565.465,E2 -8565.465} C_VEL
LIN {X 0,Y 450.097,Z 298.119,A -85,B 0,C 180,E1 -8565.887,E2 -8565.887} C_VEL
LIN {X 0,Y 450.295,Z 282.101,A -85,B 0,C 180,E1 -8566.2,E2 -8566.2} C_VEL
LIN {X 0,Y 450.902,Z 204.897,A -85,B 0,C 180,E1 -8567.436,E2 -8567.436} C_VEL
LIN {X 0,Y 447.638,Z 187.008,A -85,B 0,C 180,E1 -8567.883,E2 -8567.883} C_VEL
LIN {X 0,Y 447.628,Z 185.569,A -85,B 0,C 180,E1 -8568.088,E2 -8568.088} C_VEL
LIN {X 0,Y 448.418,Z 169.633,A -85,B 0,C 180,E1 -8571.37,E2 -8571.37} C_VEL
LIN {X 0,Y 447.446,Z 162.9,A -85,B 0,C 180,E1 -8572.852,E2 -8572.852} C_VEL
LIN {X 0,Y 446.488,Z 157.958,A -85,B 0,C 180,E1 -8574.02,E2 -8574.02} C_VEL
LIN {X 0,Y 446.476,Z 157.87,A -85,B 0,C 180,E1 -8577.161,E2 -8577.161} C_VEL
LIN {X 0,Y 446.428,Z 157.876,A -85,B 0,C 180,E1 -8580.249,E2 -8580.249} C_VEL
LIN {X 0,Y 446.446,Z 157.872,A -85,B 0,C 180,E1 -8583.453,E2 -8583.453} C_VEL
LIN {X 0,Y 446.402,Z 157.879,A -85,B 0,C 180,E1 -8586.745,E2 -8586.745} C_VEL
LIN {X 0,Y 446.44,Z 157.862,A -85,B 0,C 180,E1 -8590.198,E2 -8590.198} C_VEL
LIN {X 0,Y 446.427,Z 157.876,A -85,B 0,C 180,E1 -8592.604,E2 -8592.604} C_VEL
LIN {X 0,Y 446.448,Z 157.865,A -85,B 0,C 180,E1 -8595.103,E2 -8595.103} C_VEL
LIN {X 0,Y 446.425,Z 157.872,A -85,B 0,C 180,E1 -8598.608,E2 -8598.608} C_VEL
LIN {X 0,Y 446.456,Z 157.869,A -85,B 0,C 180,E1 -8600.974,E2 -8600.974} C_VEL
LIN {X 0,Y 446.417,Z 157.852,A -85,B 0,C 180,E1 -8604.373,E2 -8604.373} C_VEL
LIN {X 0,Y 446.418,Z 157.869,A -85,B 0,C 180,E1 -8607.638,E2 -8607.638} C_VEL
LIN {X 0,Y 446.443,Z 157.869,A -85,B 0,C 180,E1 -8610.79,E2 -8610.79} C_VEL
LIN {X 0,Y 446.473,Z 157.869,A -85,B 0,C 180,E1 -8613.848,E2 -8613.848} C_VEL
LIN {X 0,Y 446.42,Z 157.871,A -85,B 0,C 180,E1 -8616.823,E2 -8616.823} C_VEL
LIN {X 0,Y 446.438,Z 157.873,A -85,B 0,C 180,E1 -8619.737,E2 -8619.737} C_VEL
LIN {X 0,Y 446.456,Z 157.866,A -85,B 0,C 180,E1 -8622.597,E2 -8622.597} C_VEL
LIN {X 0,Y 446.463,Z 157.864,A -85,B 0,C 180,E1 -8625.412,E2 -8625.412} C_VEL
LIN {X 0,Y 446.511,Z 157.862,A -85,B 0,C 180,E1 -8628.193,E2 -8628.193} C_VEL
LIN {X 0,Y 446.594,Z 157.852,A -85,B 0,C 180,E1 -8631.858,E2 -8631.858} C_VEL
LIN {X 0,Y 446.633,Z 157.846,A -85,B 0,C 180,E1 -8634.582,E2 -8634.582} C_VEL
LIN {X 0,Y 446.655,Z 157.839,A -85,B 0,C 180,E1 -8638.197,E2 -8638.197} C_VEL
LIN {X 0,Y 446.783,Z 157.83,A -85,B 0,C 180,E1 -8640,E2 -8640} C_VEL
LIN {X 0,Y 446.682,Z 157.839,A -85,B 0,C 180,E1 -8642.705,E2 -8642.705} C_VEL
LIN {X 0,Y 446.627,Z 157.845,A -85,B 0,C 180,E1 -8646.324,E2 -8646.324} C_VEL
LIN {X 0,Y 446.526,Z 157.863,A -85,B 0,C 180,E1 -8649.056,E2 -8649.056} C_VEL
LIN {X 0,Y 446.515,Z 157.857,A -85,B 0,C 180,E1 -8652.73,E2 -8652.73} C_VEL
LIN {X 0,Y 446.482,Z 157.863,A -85,B 0,C 180,E1 -8656.459,E2 -8656.459} C_VEL
LIN {X 0,Y 446.462,Z 157.87,A -85,B 0,C 180,E1 -8659.304,E2 -8659.304} C_VEL
LIN {X 0,Y 446.411,Z 157.873,A -85,B 0,C 180,E1 -8662.2,E2 -8662.2} C_VEL
LIN {X 0,Y 446.438,Z 157.872,A -85,B 0,C 180,E1 -8665.154,E2 -8665.154} C_VEL
LIN {X 0,Y 446.48,Z 157.864,A -85,B 0,C 180,E1 -8668.179,E2 -8668.179} C_VEL
LIN {X 0,Y 446.413,Z 157.876,A -85,B 0,C 180,E1 -8671.775,E2 -8671.775} C_VEL
LIN {X 0,Y 446.418,Z 157.871,A -85,B 0,C 180,E1 -8674.524,E2 -8674.524} C_VEL
LIN {X 0,Y 446.41,Z 157.865,A -85,B 0,C 180,E1 -8678.079,E2 -8678.079} C_VEL
LIN {X 0,Y 446.419,Z 157.88,A -85,B 0,C 180,E1 -8680.917,E2 -8680.917} C_VEL
LIN {X 0,Y 446.395,Z 157.875,A -85,B 0,C 180,E1 -8683.847,E2 -8683.847} C_VEL
LIN {X 0,Y 446.39,Z 157.879,A -85,B 0,C 180,E1 -8686.405,E2 -8686.405} C_VEL
LIN {X 0,Y 446.398,Z 157.875,A -85,B 0,C 180,E1 -8689.798,E2 -8689.798} C_VEL
LIN {X 0,Y 446.403,Z 157.866,A -85,B 0,C 180,E1 -8692.121,E2 -8692.121} C_VEL
LIN {X 0,Y 446.427,Z 157.868,A -85,B 0,C 180,E1 -8695.477,E2 -8695.477} C_VEL
LIN {X 0,Y 446.415,Z 157.876,A -85,B 0,C 180,E1 -8698.7,E2 -8698.7} C_VEL
LIN {X 0,Y 446.449,Z 157.866,A -85,B 0,C 180,E1 -8701.831,E2 -8701.831} C_VEL
LIN {X 0,Y 446.494,Z 158.019,A -85,B 0,C 180,E1 -8704.726,E2 -8704.726} C_VEL
LIN {X 0,Y 448.716,Z 169.763,A -85,B 0,C 180,E1 -8707.302,E2 -8707.302} C_VEL
LIN {X 0,Y 448.076,Z 182.335,A -85,B 0,C 180,E1 -8709.814,E2 -8709.814} C_VEL
LIN {X 0,Y 447.556,Z 194.38,A -85,B 0,C 180,E1 -8712.144,E2 -8712.144} C_VEL
LIN {X 0,Y 450.848,Z 213.598,A -85,B 0,C 180,E1 -8712.621,E2 -8712.621} C_VEL
LIN {X 0,Y 450.151,Z 301.991,A -85,B 0,C 180,E1 -8714.057,E2 -8714.057} C_VEL
LIN {X 0,Y 449.688,Z 315.237,A -85,B 0,C 180,E1 -8714.447,E2 -8714.447} C_VEL
LIN {X 0,Y 449.209,Z 328.499,A -85,B 0,C 180,E1 -8715.04,E2 -8715.04} C_VEL
LIN {X 0,Y 448.667,Z 339.628,A -85,B 0,C 180,E1 -8715.717,E2 -8715.717} C_VEL
LIN {X 0,Y 448.093,Z 349.972,A -85,B 0,C 180,E1 -8716.514,E2 -8716.514} C_VEL
LIN {X 0,Y 447.551,Z 360.553,A -85,B 0,C 180,E1 -8717.53,E2 -8717.53} C_VEL
LIN {X 0,Y 446.914,Z 370.138,A -85,B 0,C 180,E1 -8718.663,E2 -8718.663} C_VEL
LIN {X 0,Y 446.507,Z 377.994,A -85,B 0,C 180,E1 -8719.8,E2 -8719.8} C_VEL
LIN {X 0,Y 446.041,Z 385.664,A -85,B 0,C 180,E1 -8721.163,E2 -8721.163} C_VEL
LIN {X 0,Y 445.676,Z 392.733,A -85,B 0,C 180,E1 -8722.752,E2 -8722.752} C_VEL
LIN {X 0,Y 445.529,Z 397.435,A -85,B 0,C 180,E1 -8724.115,E2 -8724.115} C_VEL
LIN {X 0,Y 445.416,Z 401.026,A -85,B 0,C 180,E1 -8725.475,E2 -8725.475} C_VEL
LIN {X 0,Y 445.379,Z 402.878,A -85,B 0,C 180,E1 -8726.381,E2 -8726.381} C_VEL
LIN {X 0,Y 445.403,Z 404.267,A -85,B 0,C 180,E1 -8727.286,E2 -8727.286} C_VEL
LIN {X 0,Y 445.315,Z 405.862,A -85,B 0,C 180,E1 -8729.095,E2 -8729.095} C_VEL
LIN {X 0,Y 445.316,Z 406.077,A -85,B 0,C 180,E1 -8730,E2 -8730} C_VEL
LIN {X 0,Y 445.352,Z 405.257,A -85,B 0,C 180,E1 -8731.808,E2 -8731.808} C_VEL
LIN {X 0,Y 445.403,Z 404.267,A -85,B 0,C 180,E1 -8732.713,E2 -8732.713} C_VEL
LIN {X 0,Y 445.379,Z 402.878,A -85,B 0,C 180,E1 -8733.618,E2 -8733.618} C_VEL
LIN {X 0,Y 445.489,Z 399.956,A -85,B 0,C 180,E1 -8734.977,E2 -8734.977} C_VEL
LIN {X 0,Y 445.58,Z 395.652,A -85,B 0,C 180,E1 -8736.443,E2 -8736.443} C_VEL
LIN {X 0,Y 445.816,Z 389.913,A -85,B 0,C 180,E1 -8737.928,E2 -8737.928} C_VEL
LIN {X 0,Y 446.145,Z 383.26,A -85,B 0,C 180,E1 -8739.291,E2 -8739.291} C_VEL
LIN {X 0,Y 446.631,Z 375.003,A -85,B 0,C 180,E1 -8740.654,E2 -8740.654} C_VEL
LIN {X 0,Y 447.173,Z 366.538,A -85,B 0,C 180,E1 -8741.789,E2 -8741.789} C_VEL
LIN {X 0,Y 447.793,Z 356.862,A -85,B 0,C 180,E1 -8742.845,E2 -8742.845} C_VEL
LIN {X 0,Y 448.308,Z 345.717,A -85,B 0,C 180,E1 -8743.831,E2 -8743.831} C_VEL
LIN {X 0,Y 448.881,Z 334.36,A -85,B 0,C 180,E1 -8744.623,E2 -8744.623} C_VEL
LIN {X 0,Y 449.429,Z 322.704,A -85,B 0,C 180,E1 -8745.242,E2 -8745.242} C_VEL
LIN {X 0,Y 449.904,Z 309.265,A -85,B 0,C 180,E1 -8745.748,E2 -8745.748} C_VEL
LIN {X 0,Y 450.217,Z 295.969,A -85,B 0,C 180,E1 -8746.056,E2 -8746.056} C_VEL
LIN {X 0,Y 450.841,Z 213.508,A -85,B 0,C 180,E1 -8747.377,E2 -8747.377} C_VEL
LIN {X 0,Y 447.57,Z 194.587,A -85,B 0,C 180,E1 -8747.836,E2 -8747.836} C_VEL
LIN {X 0,Y 447.635,Z 191.843,A -85,B 0,C 180,E1 -8748.3,E2 -8748.3} C_VEL
LIN {X 0,Y 448.512,Z 175.162,A -85,B 0,C 180,E1 -8751.606,E2 -8751.606} C_VEL
LIN {X 0,Y 448.683,Z 169.75,A -85,B 0,C 180,E1 -8752.696,E2 -8752.696} C_VEL
LIN {X 0,Y 446.492,Z 158.008,A -85,B 0,C 180,E1 -8755.274,E2 -8755.274} C_VEL
LIN {X 0,Y 446.438,Z 157.868,A -85,B 0,C 180,E1 -8758.181,E2 -8758.181} C_VEL
LIN {X 0,Y 446.412,Z 157.877,A -85,B 0,C 180,E1 -8761.299,E2 -8761.299} C_VEL
LIN {X 0,Y 446.424,Z 157.869,A -85,B 0,C 180,E1 -8764.522,E2 -8764.522} C_VEL
LIN {X 0,Y 446.406,Z 157.864,A -85,B 0,C 180,E1 -8768.077,E2 -8768.077} C_VEL
LIN {X 0,Y 446.412,Z 157.878,A -85,B 0,C 180,E1 -8771.391,E2 -8771.391} C_VEL
LIN {X 0,Y 446.446,Z 157.876,A -85,B 0,C 180,E1 -8775.102,E2 -8775.102} C_VEL
LIN {X 0,Y 446.42,Z 157.875,A -85,B 0,C 180,E1 -8778.608,E2 -8778.608} C_VEL
LIN {X 0,Y 446.433,Z 157.87,A -85,B 0,C 180,E1 -8780.972,E2 -8780.972} C_VEL
LIN {X 0,Y 446.41,Z 157.859,A -85,B 0,C 180,E1 -8784.373,E2 -8784.373} C_VEL
LIN {X 0,Y 446.41,Z 157.876,A -85,B 0,C 180,E1 -8787.637,E2 -8787.637} C_VEL
LIN {X 0,Y 446.436,Z 157.871,A -85,B 0,C 180,E1 -8790.79,E2 -8790.79} C_VEL
LIN {X 0,Y 446.467,Z 157.867,A -85,B 0,C 180,E1 -8793.848,E2 -8793.848} C_VEL
LIN {X 0,Y 446.414,Z 157.874,A -85,B 0,C 180,E1 -8796.822,E2 -8796.822} C_VEL
LIN {X 0,Y 446.432,Z 157.871,A -85,B 0,C 180,E1 -8799.737,E2 -8799.737} C_VEL
LIN {X 0,Y 446.444,Z 157.867,A -85,B 0,C 180,E1 -8802.596,E2 -8802.596} C_VEL
LIN {X 0,Y 446.457,Z 157.869,A -85,B 0,C 180,E1 -8805.412,E2 -8805.412} C_VEL
LIN {X 0,Y 446.529,Z 157.857,A -85,B 0,C 180,E1 -8808.193,E2 -8808.193} C_VEL
LIN {X 0,Y 446.588,Z 157.853,A -85,B 0,C 180,E1 -8811.858,E2 -8811.858} C_VEL
LIN {X 0,Y 446.627,Z 157.845,A -85,B 0,C 180,E1 -8814.582,E2 -8814.582} C_VEL
LIN {X 0,Y 446.652,Z 157.846,A -85,B 0,C 180,E1 -8818.197,E2 -8818.197} C_VEL
LIN {X 0,Y 446.779,Z 157.83,A -85,B 0,C 180,E1 -8820,E2 -8820} C_VEL
LIN {X 0,Y 446.677,Z 157.838,A -85,B 0,C 180,E1 -8822.706,E2 -8822.706} C_VEL
LIN {X 0,Y 446.625,Z 157.853,A -85,B 0,C 180,E1 -8826.324,E2 -8826.324} C_VEL
LIN {X 0,Y 446.525,Z 157.851,A -85,B 0,C 180,E1 -8829.056,E2 -8829.056} C_VEL
LIN {X 0,Y 446.509,Z 157.864,A -85,B 0,C 180,E1 -8832.73,E2 -8832.73} C_VEL
LIN {X 0,Y 446.484,Z 157.862,A -85,B 0,C 180,E1 -8836.228,E2 -8836.228} C_VEL
LIN {X 0,Y 446.458,Z 157.868,A -85,B 0,C 180,E1 -8839.304,E2 -8839.304} C_VEL
LIN {X 0,Y 446.408,Z 157.873,A -85,B 0,C 180,E1 -8842.2,E2 -8842.2} C_VEL
LIN {X 0,Y 446.447,Z 157.87,A -85,B 0,C 180,E1 -8845.153,E2 -8845.153} C_VEL
LIN {X 0,Y 446.475,Z 157.866,A -85,B 0,C 180,E1 -8848.179,E2 -8848.179} C_VEL
LIN {X 0,Y 446.409,Z 157.878,A -85,B 0,C 180,E1 -8851.776,E2 -8851.776} C_VEL
LIN {X 0,Y 446.421,Z 157.853,A -85,B 0,C 180,E1 -8854.524,E2 -8854.524} C_VEL
LIN {X 0,Y 446.408,Z 157.876,A -85,B 0,C 180,E1 -8858.08,E2 -8858.08} C_VEL
LIN {X 0,Y 446.42,Z 157.872,A -85,B 0,C 180,E1 -8860.919,E2 -8860.919} C_VEL
LIN {X 0,Y 446.391,Z 157.866,A -85,B 0,C 180,E1 -8863.848,E2 -8863.848} C_VEL
LIN {X 0,Y 446.39,Z 157.88,A -85,B 0,C 180,E1 -8866.405,E2 -8866.405} C_VEL
LIN {X 0,Y 446.421,Z 157.868,A -85,B 0,C 180,E1 -8869.084,E2 -8869.084} C_VEL
LIN {X 0,Y 446.404,Z 157.881,A -85,B 0,C 180,E1 -8872.122,E2 -8872.122} C_VEL
LIN {X 0,Y 446.426,Z 157.868,A -85,B 0,C 180,E1 -8875.478,E2 -8875.478} C_VEL
LIN {X 0,Y 446.413,Z 157.869,A -85,B 0,C 180,E1 -8878.701,E2 -8878.701} C_VEL
LIN {X 0,Y 446.483,Z 157.867,A -85,B 0,C 180,E1 -8881.822,E2 -8881.822} C_VEL
LIN {X 0,Y 446.449,Z 157.875,A -85,B 0,C 180,E1 -8884.848,E2 -8884.848} C_VEL
LIN {X 0,Y 446.507,Z 158.09,A -85,B 0,C 180,E1 -8886.132,E2 -8886.132} C_VEL
LIN {X 0,Y 448.334,Z 168.041,A -85,B 0,C 180,E1 -8888.385,E2 -8888.385} C_VEL
LIN {X 0,Y 448.037,Z 176.34,A -85,B 0,C 180,E1 -8890.113,E2 -8890.113} C_VEL
LIN {X 0,Y 447.587,Z 186.643,A -85,B 0,C 180,E1 -8892.183,E2 -8892.183} C_VEL
LIN {X 0,Y 448.486,Z 191.632,A -85,B 0,C 180,E1 -8892.344,E2 -8892.344} C_VEL
LIN {X 0,Y 450.914,Z 205.488,A -85,B 0,C 180,E1 -8892.669,E2 -8892.669} C_VEL
LIN {X 0,Y 450.44,Z 271.293,A -85,B 0,C 180,E1 -8893.724,E2 -8893.724} C_VEL
LIN {X 0,Y 449.607,Z 277.143,A -85,B 0,C 180,E1 -8893.785,E2 -8893.785} C_VEL
LIN {X 0,Y 443.868,Z 296.09,A -85,B 0,C 180,E1 -8893.923,E2 -8893.923} C_VEL
LIN {X 0,Y 443.162,Z 301.833,A -85,B 0,C 180,E1 -8894.065,E2 -8894.065} C_VEL
LIN {X 0,Y 442.702,Z 315.133,A -85,B 0,C 180,E1 -8894.58,E2 -8894.58} C_VEL
LIN {X 0,Y 442.181,Z 325.774,A -85,B 0,C 180,E1 -8895.151,E2 -8895.151} C_VEL
LIN {X 0,Y 441.568,Z 337.268,A -85,B 0,C 180,E1 -8895.954,E2 -8895.954} C_VEL
LIN {X 0,Y 441.073,Z 348.229,A -85,B 0,C 180,E1 -8896.93,E2 -8896.93} C_VEL
LIN {X 0,Y 440.38,Z 358.223,A -85,B 0,C 180,E1 -8898.027,E2 -8898.027} C_VEL
LIN {X 0,Y 439.789,Z 366.747,A -85,B 0,C 180,E1 -8899.178,E2 -8899.178} C_VEL
LIN {X 0,Y 439.301,Z 375.029,A -85,B 0,C 180,E1 -8900.563,E2 -8900.563} C_VEL
LIN {X 0,Y 438.873,Z 381.703,A -85,B 0,C 180,E1 -8901.946,E2 -8901.946} C_VEL
LIN {X 0,Y 438.634,Z 387.82,A -85,B 0,C 180,E1 -8903.561,E2 -8903.561} C_VEL
LIN {X 0,Y 438.46,Z 391.793,A -85,B 0,C 180,E1 -8904.943,E2 -8904.943} C_VEL
LIN {X 0,Y 438.34,Z 394.73,A -85,B 0,C 180,E1 -8906.323,E2 -8906.323} C_VEL
LIN {X 0,Y 438.356,Z 396.138,A -85,B 0,C 180,E1 -8907.244,E2 -8907.244} C_VEL
LIN {X 0,Y 438.231,Z 397.758,A -85,B 0,C 180,E1 -8909.082,E2 -8909.082} C_VEL
LIN {X 0,Y 438.229,Z 397.994,A -85,B 0,C 180,E1 -8910,E2 -8910} C_VEL
LIN {X 0,Y 438.231,Z 397.806,A -85,B 0,C 180,E1 -8910.919,E2 -8910.919} C_VEL
LIN {X 0,Y 438.356,Z 396.249,A -85,B 0,C 180,E1 -8912.757,E2 -8912.757} C_VEL
LIN {X 0,Y 438.337,Z 394.888,A -85,B 0,C 180,E1 -8913.677,E2 -8913.677} C_VEL
LIN {X 0,Y 438.457,Z 392.011,A -85,B 0,C 180,E1 -8915.058,E2 -8915.058} C_VEL
LIN {X 0,Y 438.641,Z 387.618,A -85,B 0,C 180,E1 -8916.595,E2 -8916.595} C_VEL
LIN {X 0,Y 438.809,Z 383.081,A -85,B 0,C 180,E1 -8917.825,E2 -8917.825} C_VEL
LIN {X 0,Y 439.213,Z 376.751,A -85,B 0,C 180,E1 -8919.208,E2 -8919.208} C_VEL
LIN {X 0,Y 439.7,Z 368.828,A -85,B 0,C 180,E1 -8920.592,E2 -8920.592} C_VEL
LIN {X 0,Y 440.323,Z 358.974,A -85,B 0,C 180,E1 -8921.976,E2 -8921.976} C_VEL
LIN {X 0,Y 440.965,Z 349.407,A -85,B 0,C 180,E1 -8923.05,E2 -8923.05} C_VEL
LIN {X 0,Y 441.505,Z 338.404,A -85,B 0,C 180,E1 -8924.049,E2 -8924.049} C_VEL
LIN {X 0,Y 442.139,Z 327.21,A -85,B 0,C 180,E1 -8924.852,E2 -8924.852} C_VEL
LIN {X 0,Y 442.689,Z 315.859,A -85,B 0,C 180,E1 -8925.481,E2 -8925.481} C_VEL
LIN {X 0,Y 443.155,Z 302.928,A -85,B 0,C 180,E1 -8925.995,E2 -8925.995} C_VEL
LIN {X 0,Y 443.488,Z 289.117,A -85,B 0,C 180,E1 -8926.337,E2 -8926.337} C_VEL
LIN {X 0,Y 444.173,Z 206.072,A -85,B 0,C 180,E1 -8927.69,E2 -8927.69} C_VEL
LIN {X 0,Y 440.715,Z 187.231,A -85,B 0,C 180,E1 -8928.165,E2 -8928.165} C_VEL
LIN {X 0,Y 440.67,Z 186.22,A -85,B 0,C 180,E1 -8928.275,E2 -8928.275} C_VEL
LIN {X 0,Y 441.485,Z 170.823,A -85,B 0,C 180,E1 -8931.477,E2 -8931.477} C_VEL
LIN {X 0,Y 440.211,Z 162.829,A -85,B 0,C 180,E1 -8933.274,E2 -8933.274} C_VEL
LIN {X 0,Y 439.42,Z 158.802,A -85,B 0,C 180,E1 -8934.265,E2 -8934.265} C_VEL
LIN {X 0,Y 439.443,Z 158.747,A -85,B 0,C 180,E1 -8937.632,E2 -8937.632} C_VEL
LIN {X 0,Y 439.362,Z 158.749,A -85,B 0,C 180,E1 -8940.788,E2 -8940.788} C_VEL
LIN {X 0,Y 439.388,Z 158.75,A -85,B 0,C 180,E1 -8944.043,E2 -8944.043} C_VEL
LIN {X 0,Y 439.349,Z 158.757,A -85,B 0,C 180,E1 -8946.887,E2 -8946.887} C_VEL
LIN {X 0,Y 439.401,Z 158.739,A -85,B 0,C 180,E1 -8949.849,E2 -8949.849} C_VEL
LIN {X 0,Y 439.379,Z 158.753,A -85,B 0,C 180,E1 -8952.626,E2 -8952.626} C_VEL
LIN {X 0,Y 439.397,Z 158.744,A -85,B 0,C 180,E1 -8955.27,E2 -8955.27} C_VEL
LIN {X 0,Y 439.386,Z 158.748,A -85,B 0,C 180,E1 -8958.743,E2 -8958.743} C_VEL
LIN {X 0,Y 439.374,Z 158.754,A -85,B 0,C 180,E1 -8961.607,E2 -8961.607} C_VEL
LIN {X 0,Y 439.396,Z 158.722,A -85,B 0,C 180,E1 -8964.844,E2 -8964.844} C_VEL
LIN {X 0,Y 439.368,Z 158.755,A -85,B 0,C 180,E1 -8968.139,E2 -8968.139} C_VEL
LIN {X 0,Y 439.428,Z 158.747,A -85,B 0,C 180,E1 -8971.598,E2 -8971.598} C_VEL
LIN {X 0,Y 439.392,Z 158.751,A -85,B 0,C 180,E1 -8974.414,E2 -8974.414} C_VEL
LIN {X 0,Y 439.358,Z 158.753,A -85,B 0,C 180,E1 -8977.424,E2 -8977.424} C_VEL
LIN {X 0,Y 439.436,Z 158.743,A -85,B 0,C 180,E1 -8980.663,E2 -8980.663} C_VEL
LIN {X 0,Y 439.456,Z 158.735,A -85,B 0,C 180,E1 -8984.224,E2 -8984.224} C_VEL
LIN {X 0,Y 439.477,Z 158.74,A -85,B 0,C 180,E1 -8988.001,E2 -8988.001} C_VEL
LIN {X 0,Y 439.541,Z 158.728,A -85,B 0,C 180,E1 -8991.726,E2 -8991.726} C_VEL
LIN {X 0,Y 439.608,Z 158.721,A -85,B 0,C 180,E1 -8994.496,E2 -8994.496} C_VEL
LIN {X 0,Y 439.625,Z 158.715,A -85,B 0,C 180,E1 -8998.168,E2 -8998.168} C_VEL
LIN {X 0,Y 439.753,Z 158.706,A -85,B 0,C 180,E1 -9000,E2 -9000} C_VEL
LIN {X 0,Y 439.632,Z 158.718,A -85,B 0,C 180,E1 -9002.749,E2 -9002.749} C_VEL
LIN {X 0,Y 439.597,Z 158.721,A -85,B 0,C 180,E1 -9006.426,E2 -9006.426} C_VEL
LIN {X 0,Y 439.489,Z 158.742,A -85,B 0,C 180,E1 -9009.202,E2 -9009.202} C_VEL
LIN {X 0,Y 439.459,Z 158.738,A -85,B 0,C 180,E1 -9012.938,E2 -9012.938} C_VEL
LIN {X 0,Y 439.44,Z 158.74,A -85,B 0,C 180,E1 -9016.348,E2 -9016.348} C_VEL
LIN {X 0,Y 439.396,Z 158.751,A -85,B 0,C 180,E1 -9019.627,E2 -9019.627} C_VEL
LIN {X 0,Y 439.357,Z 158.753,A -85,B 0,C 180,E1 -9022.576,E2 -9022.576} C_VEL
LIN {X 0,Y 439.392,Z 158.752,A -85,B 0,C 180,E1 -9025.586,E2 -9025.586} C_VEL
LIN {X 0,Y 439.412,Z 158.747,A -85,B 0,C 180,E1 -9028.674,E2 -9028.674} C_VEL
LIN {X 0,Y 439.363,Z 158.753,A -85,B 0,C 180,E1 -9032.03,E2 -9032.03} C_VEL
LIN {X 0,Y 439.387,Z 158.735,A -85,B 0,C 180,E1 -9035.34,E2 -9035.34} C_VEL
LIN {X 0,Y 439.372,Z 158.744,A -85,B 0,C 180,E1 -9038.596,E2 -9038.596} C_VEL
LIN {X 0,Y 439.378,Z 158.753,A -85,B 0,C 180,E1 -9041.256,E2 -9041.256} C_VEL
LIN {X 0,Y 439.395,Z 158.752,A -85,B 0,C 180,E1 -9044.73,E2 -9044.73} C_VEL
LIN {X 0,Y 439.356,Z 158.753,A -85,B 0,C 180,E1 -9047.792,E2 -9047.792} C_VEL
LIN {X 0,Y 439.356,Z 158.753,A -85,B 0,C 180,E1 -9050.22,E2 -9050.22} C_VEL
LIN {X 0,Y 439.371,Z 158.754,A -85,B 0,C 180,E1 -9053.713,E2 -9053.713} C_VEL
LIN {X 0,Y 439.372,Z 158.754,A -85,B 0,C 180,E1 -9057.054,E2 -9057.054} C_VEL
LIN {X 0,Y 439.377,Z 158.752,A -85,B 0,C 180,E1 -9060.274,E2 -9060.274} C_VEL
LIN {X 0,Y 439.382,Z 158.736,A -85,B 0,C 180,E1 -9063.393,E2 -9063.393} C_VEL
LIN {X 0,Y 439.449,Z 158.875,A -85,B 0,C 180,E1 -9064.482,E2 -9064.482} C_VEL
LIN {X 0,Y 441.822,Z 171.541,A -85,B 0,C 180,E1 -9067.309,E2 -9067.309} C_VEL
LIN {X 0,Y 440.885,Z 188.227,A -85,B 0,C 180,E1 -9070.685,E2 -9070.685} C_VEL
LIN {X 0,Y 440.608,Z 194.099,A -85,B 0,C 180,E1 -9071.831,E2 -9071.831} C_VEL
LIN {X 0,Y 441.319,Z 198.528,A -85,B 0,C 180,E1 -9071.982,E2 -9071.982} C_VEL
LIN {X 0,Y 444.105,Z 214.634,A -85,B 0,C 180,E1 -9072.366,E2 -9072.366} C_VEL
LIN {X 0,Y 443.339,Z 301.938,A -85,B 0,C 180,E1 -9073.805,E2 -9073.805} C_VEL
LIN {X 0,Y 442.876,Z 315.18,A -85,B 0,C 180,E1 -9074.202,E2 -9074.202} C_VEL
LIN {X 0,Y 442.404,Z 327.321,A -85,B 0,C 180,E1 -9074.745,E2 -9074.745} C_VEL
LIN {X 0,Y 441.78,Z 339.567,A -85,B 0,C 180,E1 -9075.49,E2 -9075.49} C_VEL
LIN {X 0,Y 441.15,Z 350.606,A -85,B 0,C 180,E1 -9076.361,E2 -9076.361} C_VEL
LIN {X 0,Y 440.54,Z 361.56,A -85,B 0,C 180,E1 -9077.446,E2 -9077.446} C_VEL
LIN {X 0,Y 439.941,Z 370.075,A -85,B 0,C 180,E1 -9078.481,E2 -9078.481} C_VEL
LIN {X 0,Y 439.495,Z 377.931,A -85,B 0,C 180,E1 -9079.636,E2 -9079.636} C_VEL
LIN {X 0,Y 439.017,Z 385.6,A -85,B 0,C 180,E1 -9081.02,E2 -9081.02} C_VEL
LIN {X 0,Y 438.613,Z 392.669,A -85,B 0,C 180,E1 -9082.635,E2 -9082.635} C_VEL
LIN {X 0,Y 438.452,Z 396.993,A -85,B 0,C 180,E1 -9083.897,E2 -9083.897} C_VEL
LIN {X 0,Y 438.346,Z 400.962,A -85,B 0,C 180,E1 -9085.402,E2 -9085.402} C_VEL
LIN {X 0,Y 438.281,Z 402.814,A -85,B 0,C 180,E1 -9086.322,E2 -9086.322} C_VEL
LIN {X 0,Y 438.3,Z 404.202,A -85,B 0,C 180,E1 -9087.242,E2 -9087.242} C_VEL
LIN {X 0,Y 438.274,Z 405.193,A -85,B 0,C 180,E1 -9088.162,E2 -9088.162} C_VEL
LIN {X 0,Y 438.228,Z 406.012,A -85,B 0,C 180,E1 -9090,E2 -9090} C_VEL
LIN {X 0,Y 438.274,Z 405.192,A -85,B 0,C 180,E1 -9091.837,E2 -9091.837} C_VEL
LIN {X 0,Y 438.3,Z 404.202,A -85,B 0,C 180,E1 -9092.757,E2 -9092.757} C_VEL
LIN {X 0,Y 438.281,Z 402.812,A -85,B 0,C 180,E1 -9093.677,E2 -9093.677} C_VEL
LIN {X 0,Y 438.422,Z 399.89,A -85,B 0,C 180,E1 -9095.058,E2 -9095.058} C_VEL
LIN {X 0,Y 438.505,Z 395.933,A -85,B 0,C 180,E1 -9096.441,E2 -9096.441} C_VEL
LIN {X 0,Y 438.752,Z 389.846,A -85,B 0,C 180,E1 -9098.056,E2 -9098.056} C_VEL
LIN {X 0,Y 439.12,Z 383.193,A -85,B 0,C 180,E1 -9099.441,E2 -9099.441} C_VEL
LIN {X 0,Y 439.608,Z 374.936,A -85,B 0,C 180,E1 -9100.826,E2 -9100.826} C_VEL
LIN {X 0,Y 440.206,Z 366.47,A -85,B 0,C 180,E1 -9101.978,E2 -9101.978} C_VEL
LIN {X 0,Y 440.841,Z 356.956,A -85,B 0,C 180,E1 -9103.035,E2 -9103.035} C_VEL
LIN {X 0,Y 441.322,Z 347.075,A -85,B 0,C 180,E1 -9103.937,E2 -9103.937} C_VEL
LIN {X 0,Y 441.899,Z 336.058,A -85,B 0,C 180,E1 -9104.741,E2 -9104.741} C_VEL
LIN {X 0,Y 442.537,Z 323.845,A -85,B 0,C 180,E1 -9105.426,E2 -9105.426} C_VEL
LIN {X 0,Y 443.018,Z 311.021,A -85,B 0,C 180,E1 -9105.94,E2 -9105.94} C_VEL
LIN {X 0,Y 443.397,Z 297.41,A -85,B 0,C 180,E1 -9106.28,E2 -9106.28} C_VEL
LIN {X 0,Y 444.073,Z 214.523,A -85,B 0,C 180,E1 -9107.632,E2 -9107.632} C_VEL
LIN {X 0,Y 440.614,Z 194.465,A -85,B 0,C 180,E1 -9108.131,E2 -9108.131} C_VEL
LIN {X 0,Y 440.768,Z 190.585,A -85,B 0,C 180,E1 -9108.837,E2 -9108.837} C_VEL
LIN {X 0,Y 441.737,Z 173.903,A -85,B 0,C 180,E1 -9112.2,E2 -9112.2} C_VEL
LIN {X 0,Y 441.583,Z 170.096,A -85,B 0,C 180,E1 -9112.996,E2 -9112.996} C_VEL
LIN {X 0,Y 439.447,Z 158.862,A -85,B 0,C 180,E1 -9115.518,E2 -9115.518} C_VEL
LIN {X 0,Y 439.394,Z 158.749,A -85,B 0,C 180,E1 -9118.674,E2 -9118.674} C_VEL
LIN {X 0,Y 439.366,Z 158.755,A -85,B 0,C 180,E1 -9122.029,E2 -9122.029} C_VEL
LIN {X 0,Y 439.389,Z 158.755,A -85,B 0,C 180,E1 -9125.339,E2 -9125.339} C_VEL
LIN {X 0,Y 439.358,Z 158.742,A -85,B 0,C 180,E1 -9128.596,E2 -9128.596} C_VEL
LIN {X 0,Y 439.375,Z 158.757,A -85,B 0,C 180,E1 -9131.254,E2 -9131.254} C_VEL
LIN {X 0,Y 439.394,Z 158.752,A -85,B 0,C 180,E1 -9134.728,E2 -9134.728} C_VEL
LIN {X 0,Y 439.388,Z 158.749,A -85,B 0,C 180,E1 -9137.795,E2 -9137.795} C_VEL
LIN {X 0,Y 439.388,Z 158.749,A -85,B 0,C 180,E1 -9140.223,E2 -9140.223} C_VEL
LIN {X 0,Y 439.364,Z 158.735,A -85,B 0,C 180,E1 -9143.712,E2 -9143.712} C_VEL
LIN {X 0,Y 439.363,Z 158.758,A -85,B 0,C 180,E1 -9147.053,E2 -9147.053} C_VEL
LIN {X 0,Y 439.371,Z 158.749,A -85,B 0,C 180,E1 -9150.273,E2 -9150.273} C_VEL
LIN {X 0,Y 439.417,Z 158.747,A -85,B 0,C 180,E1 -9153.395,E2 -9153.395} C_VEL
LIN {X 0,Y 439.372,Z 158.747,A -85,B 0,C 180,E1 -9156.429,E2 -9156.429} C_VEL
LIN {X 0,Y 439.376,Z 158.751,A -85,B 0,C 180,E1 -9159.396,E2 -9159.396} C_VEL
LIN {X 0,Y 439.393,Z 158.743,A -85,B 0,C 180,E1 -9162.308,E2 -9162.308} C_VEL
LIN {X 0,Y 439.434,Z 158.746,A -85,B 0,C 180,E1 -9165.174,E2 -9165.174} C_VEL
LIN {X 0,Y 439.497,Z 158.731,A -85,B 0,C 180,E1 -9168.002,E2 -9168.002} C_VEL
LIN {X 0,Y 439.536,Z 158.731,A -85,B 0,C 180,E1 -9171.726,E2 -9171.726} C_VEL
LIN {X 0,Y 439.602,Z 158.72,A -85,B 0,C 180,E1 -9174.496,E2 -9174.496} C_VEL
LIN {X 0,Y 439.622,Z 158.722,A -85,B 0,C 180,E1 -9178.168,E2 -9178.168} C_VEL
LIN {X 0,Y 439.749,Z 158.706,A -85,B 0,C 180,E1 -9180,E2 -9180} C_VEL
LIN {X 0,Y 439.626,Z 158.716,A -85,B 0,C 180,E1 -9182.749,E2 -9182.749} C_VEL
LIN {X 0,Y 439.6,Z 158.728,A -85,B 0,C 180,E1 -9186.426,E2 -9186.426} C_VEL
LIN {X 0,Y 439.487,Z 158.727,A -85,B 0,C 180,E1 -9189.202,E2 -9189.202} C_VEL
LIN {X 0,Y 439.453,Z 158.741,A -85,B 0,C 180,E1 -9192.938,E2 -9192.938} C_VEL
LIN {X 0,Y 439.436,Z 158.741,A -85,B 0,C 180,E1 -9196.349,E2 -9196.349} C_VEL
LIN {X 0,Y 439.392,Z 158.75,A -85,B 0,C 180,E1 -9199.627,E2 -9199.627} C_VEL
LIN {X 0,Y 439.355,Z 158.753,A -85,B 0,C 180,E1 -9202.576,E2 -9202.576} C_VEL
LIN {X 0,Y 439.395,Z 158.75,A -85,B 0,C 180,E1 -9205.586,E2 -9205.586} C_VEL
LIN {X 0,Y 439.407,Z 158.747,A -85,B 0,C 180,E1 -9208.674,E2 -9208.674} C_VEL
LIN {X 0,Y 439.361,Z 158.754,A -85,B 0,C 180,E1 -9212.031,E2 -9212.031} C_VEL
LIN {X 0,Y 439.387,Z 158.726,A -85,B 0,C 180,E1 -9215.341,E2 -9215.341} C_VEL
LIN {X 0,Y 439.371,Z 158.753,A -85,B 0,C 180,E1 -9218.596,E2 -9218.596} C_VEL
LIN {X 0,Y 439.381,Z 158.749,A -85,B 0,C 180,E1 -9221.258,E2 -9221.258} C_VEL
LIN {X 0,Y 439.392,Z 158.744,A -85,B 0,C 180,E1 -9224.731,E2 -9224.731} C_VEL
LIN {X 0,Y 439.39,Z 158.753,A -85,B 0,C 180,E1 -9227.797,E2 -9227.797} C_VEL
LIN {X 0,Y 439.39,Z 158.74,A -85,B 0,C 180,E1 -9230.225,E2 -9230.225} C_VEL
LIN {X 0,Y 439.371,Z 158.755,A -85,B 0,C 180,E1 -9233.714,E2 -9233.714} C_VEL
LIN {X 0,Y 439.369,Z 158.754,A -85,B 0,C 180,E1 -9237.055,E2 -9237.055} C_VEL
LIN {X 0,Y 439.38,Z 158.754,A -85,B 0,C 180,E1 -9240.275,E2 -9240.275} C_VEL
LIN {X 0,Y 439.427,Z 158.748,A -85,B 0,C 180,E1 -9243.397,E2 -9243.397} C_VEL
LIN {X 0,Y 439.447,Z 158.797,A -85,B 0,C 180,E1 -9245.834,E2 -9245.834} C_VEL
LIN {X 0,Y 440.367,Z 163.526,A -85,B 0,C 180,E1 -9246.984,E2 -9246.984} C_VEL
LIN {X 0,Y 441.484,Z 170.376,A -85,B 0,C 180,E1 -9248.523,E2 -9248.523} C_VEL
LIN {X 0,Y 440.662,Z 186.469,A -85,B 0,C 180,E1 -9251.862,E2 -9251.862} C_VEL
LIN {X 0,Y 440.758,Z 187.546,A -85,B 0,C 180,E1 -9251.943,E2 -9251.943} C_VEL
LIN {X 0,Y 444.16,Z 206.662,A -85,B 0,C 180,E1 -9252.415,E2 -9252.415} C_VEL
LIN {X 0,Y 443.384,Z 294.531,A -85,B 0,C 180,E1 -9253.867,E2 -9253.867} C_VEL
LIN {X 0,Y 443.162,Z 301.833,A -85,B 0,C 180,E1 -9254.065,E2 -9254.065} C_VEL
LIN {X 0,Y 442.733,Z 305.646,A -85,B 0,C 180,E1 -9254.179,E2 -9254.179} C_VEL
LIN {X 0,Y 440.546,Z 313.051,A -85,B 0,C 180,E1 -9254.404,E2 -9254.404} C_VEL
LIN {X 0,Y 436.21,Z 324.703,A -85,B 0,C 180,E1 -9254.874,E2 -9254.874} C_VEL
LIN {X 0,Y 435.051,Z 330.832,A -85,B 0,C 180,E1 -9255.239,E2 -9255.239} C_VEL
LIN {X 0,Y 434.444,Z 342.137,A -85,B 0,C 180,E1 -9256.132,E2 -9256.132} C_VEL
LIN {X 0,Y 433.766,Z 353.317,A -85,B 0,C 180,E1 -9257.247,E2 -9257.247} C_VEL
LIN {X 0,Y 433.173,Z 361.887,A -85,B 0,C 180,E1 -9258.3,E2 -9258.3} C_VEL
LIN {X 0,Y 432.637,Z 369.782,A -85,B 0,C 180,E1 -9259.471,E2 -9259.471} C_VEL
LIN {X 0,Y 432.115,Z 377.503,A -85,B 0,C 180,E1 -9260.876,E2 -9260.876} C_VEL
LIN {X 0,Y 431.658,Z 384.589,A -85,B 0,C 180,E1 -9262.516,E2 -9262.516} C_VEL
LIN {X 0,Y 431.522,Z 388.736,A -85,B 0,C 180,E1 -9263.734,E2 -9263.734} C_VEL
LIN {X 0,Y 431.31,Z 392.927,A -85,B 0,C 180,E1 -9265.327,E2 -9265.327} C_VEL
LIN {X 0,Y 431.243,Z 394.796,A -85,B 0,C 180,E1 -9266.263,E2 -9266.263} C_VEL
LIN {X 0,Y 431.254,Z 396.204,A -85,B 0,C 180,E1 -9267.198,E2 -9267.198} C_VEL
LIN {X 0,Y 431.149,Z 397.823,A -85,B 0,C 180,E1 -9269.066,E2 -9269.066} C_VEL
LIN {X 0,Y 431.144,Z 398.059,A -85,B 0,C 180,E1 -9270,E2 -9270} C_VEL
LIN {X 0,Y 431.149,Z 397.871,A -85,B 0,C 180,E1 -9270.934,E2 -9270.934} C_VEL
LIN {X 0,Y 431.205,Z 397.284,A -85,B 0,C 180,E1 -9271.868,E2 -9271.868} C_VEL
LIN {X 0,Y 431.254,Z 396.313,A -85,B 0,C 180,E1 -9272.803,E2 -9272.803} C_VEL
LIN {X 0,Y 431.24,Z 394.952,A -85,B 0,C 180,E1 -9273.738,E2 -9273.738} C_VEL
LIN {X 0,Y 431.396,Z 392.075,A -85,B 0,C 180,E1 -9275.141,E2 -9275.141} C_VEL
LIN {X 0,Y 431.564,Z 388.031,A -85,B 0,C 180,E1 -9276.593,E2 -9276.593} C_VEL
LIN {X 0,Y 431.762,Z 383.144,A -85,B 0,C 180,E1 -9277.953,E2 -9277.953} C_VEL
LIN {X 0,Y 432.19,Z 376.814,A -85,B 0,C 180,E1 -9279.359,E2 -9279.359} C_VEL
LIN {X 0,Y 432.705,Z 368.89,A -85,B 0,C 180,E1 -9280.765,E2 -9280.765} C_VEL
LIN {X 0,Y 433.363,Z 359.036,A -85,B 0,C 180,E1 -9282.171,E2 -9282.171} C_VEL
LIN {X 0,Y 434.04,Z 349.624,A -85,B 0,C 180,E1 -9283.247,E2 -9283.247} C_VEL
LIN {X 0,Y 434.552,Z 339.888,A -85,B 0,C 180,E1 -9284.159,E2 -9284.159} C_VEL
LIN {X 0,Y 435.166,Z 329.032,A -85,B 0,C 180,E1 -9284.975,E2 -9284.975} C_VEL
LIN {X 0,Y 435.8,Z 317.045,A -85,B 0,C 180,E1 -9285.672,E2 -9285.672} C_VEL
LIN {X 0,Y 436.326,Z 303.894,A -85,B 0,C 180,E1 -9286.222,E2 -9286.222} C_VEL
LIN {X 0,Y 436.671,Z 290.664,A -85,B 0,C 180,E1 -9286.569,E2 -9286.569} C_VEL
LIN {X 0,Y 437.37,Z 206.712,A -85,B 0,C 180,E1 -9287.964,E2 -9287.964} C_VEL
LIN {X 0,Y 433.753,Z 186.921,A -85,B 0,C 180,E1 -9288.486,E2 -9288.486} C_VEL
LIN {X 0,Y 434.015,Z 181.201,A -85,B 0,C 180,E1 -9289.634,E2 -9289.634} C_VEL
LIN {X 0,Y 434.472,Z 170.871,A -85,B 0,C 180,E1 -9291.842,E2 -9291.842} C_VEL
LIN {X 0,Y 432.396,Z 159.707,A -85,B 0,C 180,E1 -9294.481,E2 -9294.481} C_VEL
LIN {X 0,Y 432.393,Z 159.626,A -85,B 0,C 180,E1 -9297.071,E2 -9297.071} C_VEL
LIN {X 0,Y 432.348,Z 159.626,A -85,B 0,C 180,E1 -9300.51,E2 -9300.51} C_VEL
LIN {X 0,Y 432.36,Z 159.626,A -85,B 0,C 180,E1 -9304.003,E2 -9304.003} C_VEL
LIN {X 0,Y 432.322,Z 159.631,A -85,B 0,C 180,E1 -9307.196,E2 -9307.196} C_VEL
LIN {X 0,Y 432.323,Z 159.621,A -85,B 0,C 180,E1 -9310.56,E2 -9310.56} C_VEL
LIN {X 0,Y 432.315,Z 159.631,A -85,B 0,C 180,E1 -9313.061,E2 -9313.061} C_VEL
LIN {X 0,Y 432.331,Z 159.623,A -85,B 0,C 180,E1 -9315.664,E2 -9315.664} C_VEL
LIN {X 0,Y 432.33,Z 159.627,A -85,B 0,C 180,E1 -9318.397,E2 -9318.397} C_VEL
LIN {X 0,Y 432.336,Z 159.631,A -85,B 0,C 180,E1 -9321.85,E2 -9321.85} C_VEL
LIN {X 0,Y 432.337,Z 159.602,A -85,B 0,C 180,E1 -9325.322,E2 -9325.322} C_VEL
LIN {X 0,Y 432.317,Z 159.631,A -85,B 0,C 180,E1 -9328.653,E2 -9328.653} C_VEL
LIN {X 0,Y 432.377,Z 159.622,A -85,B 0,C 180,E1 -9331.876,E2 -9331.876} C_VEL
LIN {X 0,Y 432.341,Z 159.628,A -85,B 0,C 180,E1 -9334.998,E2 -9334.998} C_VEL
LIN {X 0,Y 432.352,Z 159.623,A -85,B 0,C 180,E1 -9338.045,E2 -9338.045} C_VEL
LIN {X 0,Y 432.381,Z 159.623,A -85,B 0,C 180,E1 -9341.029,E2 -9341.029} C_VEL
LIN {X 0,Y 432.424,Z 159.612,A -85,B 0,C 180,E1 -9343.961,E2 -9343.961} C_VEL
LIN {X 0,Y 432.453,Z 159.617,A -85,B 0,C 180,E1 -9347.803,E2 -9347.803} C_VEL
LIN {X 0,Y 432.486,Z 159.604,A -85,B 0,C 180,E1 -9351.59,E2 -9351.59} C_VEL
LIN {X 0,Y 432.585,Z 159.596,A -85,B 0,C 180,E1 -9354.406,E2 -9354.406} C_VEL
LIN {X 0,Y 432.595,Z 159.59,A -85,B 0,C 180,E1 -9358.138,E2 -9358.138} C_VEL
LIN {X 0,Y 432.723,Z 159.582,A -85,B 0,C 180,E1 -9360,E2 -9360} C_VEL
LIN {X 0,Y 432.583,Z 159.596,A -85,B 0,C 180,E1 -9362.794,E2 -9362.794} C_VEL
LIN {X 0,Y 432.547,Z 159.599,A -85,B 0,C 180,E1 -9366.531,E2 -9366.531} C_VEL
LIN {X 0,Y 432.433,Z 159.619,A -85,B 0,C 180,E1 -9369.353,E2 -9369.353} C_VEL
LIN {X 0,Y 432.424,Z 159.613,A -85,B 0,C 180,E1 -9372.803,E2 -9372.803} C_VEL
LIN {X 0,Y 432.406,Z 159.617,A -85,B 0,C 180,E1 -9376.479,E2 -9376.479} C_VEL
LIN {X 0,Y 432.332,Z 159.629,A -85,B 0,C 180,E1 -9379.961,E2 -9379.961} C_VEL
LIN {X 0,Y 432.311,Z 159.633,A -85,B 0,C 180,E1 -9382.965,E2 -9382.965} C_VEL
LIN {X 0,Y 432.355,Z 159.626,A -85,B 0,C 180,E1 -9386.033,E2 -9386.033} C_VEL
LIN {X 0,Y 432.337,Z 159.627,A -85,B 0,C 180,E1 -9389.188,E2 -9389.188} C_VEL
LIN {X 0,Y 432.318,Z 159.632,A -85,B 0,C 180,E1 -9392.444,E2 -9392.444} C_VEL
LIN {X 0,Y 432.339,Z 159.609,A -85,B 0,C 180,E1 -9395.632,E2 -9395.632} C_VEL
LIN {X 0,Y 432.335,Z 159.622,A -85,B 0,C 180,E1 -9398.715,E2 -9398.715} C_VEL
LIN {X 0,Y 432.321,Z 159.628,A -85,B 0,C 180,E1 -9401.799,E2 -9401.799} C_VEL
LIN {X 0,Y 432.331,Z 159.628,A -85,B 0,C 180,E1 -9404.348,E2 -9404.348} C_VEL
LIN {X 0,Y 432.304,Z 159.633,A -85,B 0,C 180,E1 -9407.018,E2 -9407.018} C_VEL
LIN {X 0,Y 432.306,Z 159.63,A -85,B 0,C 180,E1 -9409.825,E2 -9409.825} C_VEL
LIN {X 0,Y 432.303,Z 159.633,A -85,B 0,C 180,E1 -9413.022,E2 -9413.022} C_VEL
LIN {X 0,Y 432.359,Z 159.62,A -85,B 0,C 180,E1 -9415.997,E2 -9415.997} C_VEL
LIN {X 0,Y 432.346,Z 159.624,A -85,B 0,C 180,E1 -9419.49,E2 -9419.49} C_VEL
LIN {X 0,Y 432.343,Z 159.62,A -85,B 0,C 180,E1 -9421.874,E2 -9421.874} C_VEL
LIN {X 0,Y 432.401,Z 159.729,A -85,B 0,C 180,E1 -9424.229,E2 -9424.229} C_VEL
LIN {X 0,Y 434.804,Z 172.42,A -85,B 0,C 180,E1 -9427.121,E2 -9427.121} C_VEL
LIN {X 0,Y 434.259,Z 183.303,A -85,B 0,C 180,E1 -9429.371,E2 -9429.371} C_VEL
LIN {X 0,Y 433.68,Z 194.249,A -85,B 0,C 180,E1 -9431.551,E2 -9431.551} C_VEL
LIN {X 0,Y 437.338,Z 215.483,A -85,B 0,C 180,E1 -9432.099,E2 -9432.099} C_VEL
LIN {X 0,Y 436.55,Z 301.885,A -85,B 0,C 180,E1 -9433.546,E2 -9433.546} C_VEL
LIN {X 0,Y 436.055,Z 315.123,A -85,B 0,C 180,E1 -9433.948,E2 -9433.948} C_VEL
LIN {X 0,Y 435.552,Z 327.262,A -85,B 0,C 180,E1 -9434.499,E2 -9434.499} C_VEL
LIN {X 0,Y 434.888,Z 339.506,A -85,B 0,C 180,E1 -9435.254,E2 -9435.254} C_VEL
LIN {X 0,Y 434.181,Z 351.421,A -85,B 0,C 180,E1 -9436.218,E2 -9436.218} C_VEL
LIN {X 0,Y 433.597,Z 361.498,A -85,B 0,C 180,E1 -9437.241,E2 -9437.241} C_VEL
LIN {X 0,Y 432.976,Z 370.013,A -85,B 0,C 180,E1 -9438.293,E2 -9438.293} C_VEL
LIN {X 0,Y 432.464,Z 377.867,A -85,B 0,C 180,E1 -9439.466,E2 -9439.466} C_VEL
LIN {X 0,Y 431.966,Z 385.536,A -85,B 0,C 180,E1 -9440.872,E2 -9440.872} C_VEL
LIN {X 0,Y 431.547,Z 392.605,A -85,B 0,C 180,E1 -9442.514,E2 -9442.514} C_VEL
LIN {X 0,Y 431.353,Z 397.353,A -85,B 0,C 180,E1 -9443.936,E2 -9443.936} C_VEL
LIN {X 0,Y 431.28,Z 400.898,A -85,B 0,C 180,E1 -9445.326,E2 -9445.326} C_VEL
LIN {X 0,Y 431.188,Z 402.749,A -85,B 0,C 180,E1 -9446.262,E2 -9446.262} C_VEL
LIN {X 0,Y 431.197,Z 404.138,A -85,B 0,C 180,E1 -9447.197,E2 -9447.197} C_VEL
LIN {X 0,Y 431.197,Z 405.129,A -85,B 0,C 180,E1 -9448.132,E2 -9448.132} C_VEL
LIN {X 0,Y 431.144,Z 405.948,A -85,B 0,C 180,E1 -9450,E2 -9450} C_VEL
LIN {X 0,Y 431.197,Z 405.127,A -85,B 0,C 180,E1 -9451.868,E2 -9451.868} C_VEL
LIN {X 0,Y 431.197,Z 404.136,A -85,B 0,C 180,E1 -9452.802,E2 -9452.802} C_VEL
LIN {X 0,Y 431.188,Z 402.746,A -85,B 0,C 180,E1 -9453.738,E2 -9453.738} C_VEL
LIN {X 0,Y 431.336,Z 399.824,A -85,B 0,C 180,E1 -9455.141,E2 -9455.141} C_VEL
LIN {X 0,Y 431.441,Z 395.867,A -85,B 0,C 180,E1 -9456.547,E2 -9456.547} C_VEL
LIN {X 0,Y 431.708,Z 389.78,A -85,B 0,C 180,E1 -9458.189,E2 -9458.189} C_VEL
LIN {X 0,Y 432.101,Z 383.126,A -85,B 0,C 180,E1 -9459.596,E2 -9459.596} C_VEL
LIN {X 0,Y 432.61,Z 374.868,A -85,B 0,C 180,E1 -9461.004,E2 -9461.004} C_VEL
LIN {X 0,Y 433.242,Z 366.402,A -85,B 0,C 180,E1 -9462.173,E2 -9462.173} C_VEL
LIN {X 0,Y 433.929,Z 356.299,A -85,B 0,C 180,E1 -9463.306,E2 -9463.306} C_VEL
LIN {X 0,Y 434.518,Z 345.579,A -85,B 0,C 180,E1 -9464.279,E2 -9464.279} C_VEL
LIN {X 0,Y 435.16,Z 334.221,A -85,B 0,C 180,E1 -9465.094,E2 -9465.094} C_VEL
LIN {X 0,Y 435.763,Z 322.56,A -85,B 0,C 180,E1 -9465.732,E2 -9465.732} C_VEL
LIN {X 0,Y 436.281,Z 309.117,A -85,B 0,C 180,E1 -9466.253,E2 -9466.253} C_VEL
LIN {X 0,Y 436.607,Z 295.804,A -85,B 0,C 180,E1 -9466.571,E2 -9466.571} C_VEL
LIN {X 0,Y 437.309,Z 215.299,A -85,B 0,C 180,E1 -9467.899,E2 -9467.899} C_VEL
LIN {X 0,Y 433.688,Z 194.33,A -85,B 0,C 180,E1 -9468.435,E2 -9468.435} C_VEL
LIN {X 0,Y 434.084,Z 185.825,A -85,B 0,C 180,E1 -9470.108,E2 -9470.108} C_VEL
LIN {X 0,Y 434.82,Z 172.643,A -85,B 0,C 180,E1 -9472.824,E2 -9472.824} C_VEL
LIN {X 0,Y 432.597,Z 160.688,A -85,B 0,C 180,E1 -9475.499,E2 -9475.499} C_VEL
LIN {X 0,Y 432.374,Z 159.645,A -85,B 0,C 180,E1 -9475.836,E2 -9475.836} C_VEL
LIN {X 0,Y 432.329,Z 159.635,A -85,B 0,C 180,E1 -9479.187,E2 -9479.187} C_VEL
LIN {X 0,Y 432.319,Z 159.633,A -85,B 0,C 180,E1 -9482.442,E2 -9482.442} C_VEL
LIN {X 0,Y 432.339,Z 159.632,A -85,B 0,C 180,E1 -9485.63,E2 -9485.63} C_VEL
LIN {X 0,Y 432.321,Z 159.619,A -85,B 0,C 180,E1 -9488.711,E2 -9488.711} C_VEL
LIN {X 0,Y 432.318,Z 159.63,A -85,B 0,C 180,E1 -9491.797,E2 -9491.797} C_VEL
LIN {X 0,Y 432.327,Z 159.63,A -85,B 0,C 180,E1 -9494.346,E2 -9494.346} C_VEL
LIN {X 0,Y 432.313,Z 159.63,A -85,B 0,C 180,E1 -9497.015,E2 -9497.015} C_VEL
LIN {X 0,Y 432.325,Z 159.629,A -85,B 0,C 180,E1 -9499.82,E2 -9499.82} C_VEL
LIN {X 0,Y 432.297,Z 159.614,A -85,B 0,C 180,E1 -9503.021,E2 -9503.021} C_VEL
LIN {X 0,Y 432.35,Z 159.622,A -85,B 0,C 180,E1 -9505.996,E2 -9505.996} C_VEL
LIN {X 0,Y 432.337,Z 159.625,A -85,B 0,C 180,E1 -9509.489,E2 -9509.489} C_VEL
LIN {X 0,Y 432.38,Z 159.629,A -85,B 0,C 180,E1 -9512.927,E2 -9512.927} C_VEL
LIN {X 0,Y 432.356,Z 159.618,A -85,B 0,C 180,E1 -9516.022,E2 -9516.022} C_VEL
LIN {X 0,Y 432.338,Z 159.631,A -85,B 0,C 180,E1 -9519.045,E2 -9519.045} C_VEL
LIN {X 0,Y 432.349,Z 159.619,A -85,B 0,C 180,E1 -9522.01,E2 -9522.01} C_VEL
LIN {X 0,Y 432.383,Z 159.627,A -85,B 0,C 180,E1 -9524.926,E2 -9524.926} C_VEL
LIN {X 0,Y 432.469,Z 159.605,A -85,B 0,C 180,E1 -9527.804,E2 -9527.804} C_VEL
LIN {X 0,Y 432.48,Z 159.61,A -85,B 0,C 180,E1 -9531.59,E2 -9531.59} C_VEL
LIN {X 0,Y 432.579,Z 159.596,A -85,B 0,C 180,E1 -9534.406,E2 -9534.406} C_VEL
LIN {X 0,Y 432.592,Z 159.597,A -85,B 0,C 180,E1 -9538.138,E2 -9538.138} C_VEL
LIN {X 0,Y 432.719,Z 159.582,A -85,B 0,C 180,E1 -9540,E2 -9540} C_VEL
LIN {X 0,Y 432.578,Z 159.594,A -85,B 0,C 180,E1 -9542.794,E2 -9542.794} C_VEL
LIN {X 0,Y 432.555,Z 159.604,A -85,B 0,C 180,E1 -9546.531,E2 -9546.531} C_VEL
LIN {X 0,Y 432.431,Z 159.605,A -85,B 0,C 180,E1 -9549.353,E2 -9549.353} C_VEL
LIN {X 0,Y 432.419,Z 159.619,A -85,B 0,C 180,E1 -9552.804,E2 -9552.804} C_VEL
LIN {X 0,Y 432.401,Z 159.618,A -85,B 0,C 180,E1 -9556.479,E2 -9556.479} C_VEL
LIN {X 0,Y 432.328,Z 159.633,A -85,B 0,C 180,E1 -9559.961,E2 -9559.961} C_VEL
LIN {X 0,Y 432.309,Z 159.628,A -85,B 0,C 180,E1 -9562.965,E2 -9562.965} C_VEL
LIN {X 0,Y 432.355,Z 159.631,A -85,B 0,C 180,E1 -9566.033,E2 -9566.033} C_VEL
LIN {X 0,Y 432.333,Z 159.627,A -85,B 0,C 180,E1 -9569.188,E2 -9569.188} C_VEL
LIN {X 0,Y 432.314,Z 159.626,A -85,B 0,C 180,E1 -9572.444,E2 -9572.444} C_VEL
LIN {X 0,Y 432.336,Z 159.604,A -85,B 0,C 180,E1 -9575.633,E2 -9575.633} C_VEL
LIN {X 0,Y 432.339,Z 159.628,A -85,B 0,C 180,E1 -9579.344,E2 -9579.344} C_VEL
LIN {X 0,Y 432.327,Z 159.626,A -85,B 0,C 180,E1 -9581.798,E2 -9581.798} C_VEL
LIN {X 0,Y 432.327,Z 159.621,A -85,B 0,C 180,E1 -9584.348,E2 -9584.348} C_VEL
LIN {X 0,Y 432.314,Z 159.631,A -85,B 0,C 180,E1 -9587.017,E2 -9587.017} C_VEL
LIN {X 0,Y 432.328,Z 159.619,A -85,B 0,C 180,E1 -9589.822,E2 -9589.822} C_VEL
LIN {X 0,Y 432.303,Z 159.634,A -85,B 0,C 180,E1 -9593.023,E2 -9593.023} C_VEL
LIN {X 0,Y 432.356,Z 159.624,A -85,B 0,C 180,E1 -9595.998,E2 -9595.998} C_VEL
LIN {X 0,Y 432.345,Z 159.625,A -85,B 0,C 180,E1 -9599.491,E2 -9599.491} C_VEL
LIN {X 0,Y 432.39,Z 159.626,A -85,B 0,C 180,E1 -9602.929,E2 -9602.929} C_VEL
LIN {X 0,Y 432.396,Z 159.751,A -85,B 0,C 180,E1 -9605.643,E2 -9605.643} C_VEL
LIN {X 0,Y 434.414,Z 170.43,A -85,B 0,C 180,E1 -9608.156,E2 -9608.156} C_VEL
LIN {X 0,Y 434.31,Z 176.046,A -85,B 0,C 180,E1 -9609.369,E2 -9609.369} C_VEL
LIN {X 0,Y 433.729,Z 186.785,A -85,B 0,C 180,E1 -9611.596,E2 -9611.596} C_VEL
LIN {X 0,Y 434.914,Z 193.207,A -85,B 0,C 180,E1 -9611.797,E2 -9611.797} C_VEL
LIN {X 0,Y 437.389,Z 207.078,A -85,B 0,C 180,E1 -9612.139,E2 -9612.139} C_VEL
LIN {X 0,Y 436.594,Z 294.613,A -85,B 0,C 180,E1 -9613.609,E2 -9613.609} C_VEL
LIN {X 0,Y 436.193,Z 306.945,A -85,B 0,C 180,E1 -9613.984,E2 -9613.984} C_VEL
LIN {X 0,Y 435.604,Z 319.768,A -85,B 0,C 180,E1 -9614.562,E2 -9614.562} C_VEL
LIN {X 0,Y 435.051,Z 330.832,A -85,B 0,C 180,E1 -9615.239,E2 -9615.239} C_VEL
LIN {X 0,Y 434.143,Z 336.034,A -85,B 0,C 180,E1 -9615.59,E2 -9615.59} C_VEL
LIN {X 0,Y 430.962,Z 344.237,A -85,B 0,C 180,E1 -9616.197,E2 -9616.197} C_VEL
LIN {X 0,Y 427.697,Z 351.977,A -85,B 0,C 180,E1 -9616.9,E2 -9616.9} C_VEL
LIN {X 0,Y 426.668,Z 356.456,A -85,B 0,C 180,E1 -9617.4,E2 -9617.4} C_VEL
LIN {X 0,Y 425.91,Z 365.28,A -85,B 0,C 180,E1 -9618.58,E2 -9618.58} C_VEL
LIN {X 0,Y 425.349,Z 373.932,A -85,B 0,C 180,E1 -9620.01,E2 -9620.01} C_VEL
LIN {X 0,Y 424.863,Z 380.832,A -85,B 0,C 180,E1 -9621.439,E2 -9621.439} C_VEL
LIN {X 0,Y 424.537,Z 386.357,A -85,B 0,C 180,E1 -9622.868,E2 -9622.868} C_VEL
LIN {X 0,Y 424.384,Z 390.696,A -85,B 0,C 180,E1 -9624.298,E2 -9624.298} C_VEL
LIN {X 0,Y 424.247,Z 392.992,A -85,B 0,C 180,E1 -9625.249,E2 -9625.249} C_VEL
LIN {X 0,Y 424.151,Z 394.862,A -85,B 0,C 180,E1 -9626.2,E2 -9626.2} C_VEL
LIN {X 0,Y 424.153,Z 396.269,A -85,B 0,C 180,E1 -9627.151,E2 -9627.151} C_VEL
LIN {X 0,Y 424.131,Z 397.271,A -85,B 0,C 180,E1 -9628.101,E2 -9628.101} C_VEL
LIN {X 0,Y 424.062,Z 398.123,A -85,B 0,C 180,E1 -9630,E2 -9630} C_VEL
LIN {X 0,Y 424.07,Z 397.935,A -85,B 0,C 180,E1 -9630.95,E2 -9630.95} C_VEL
LIN {X 0,Y 424.132,Z 397.348,A -85,B 0,C 180,E1 -9631.9,E2 -9631.9} C_VEL
LIN {X 0,Y 424.152,Z 396.378,A -85,B 0,C 180,E1 -9632.85,E2 -9632.85} C_VEL
LIN {X 0,Y 424.148,Z 395.017,A -85,B 0,C 180,E1 -9633.801,E2 -9633.801} C_VEL
LIN {X 0,Y 424.316,Z 392.139,A -85,B 0,C 180,E1 -9635.227,E2 -9635.227} C_VEL
LIN {X 0,Y 424.502,Z 388.239,A -85,B 0,C 180,E1 -9636.655,E2 -9636.655} C_VEL
LIN {X 0,Y 424.714,Z 383.208,A -85,B 0,C 180,E1 -9638.086,E2 -9638.086} C_VEL
LIN {X 0,Y 425.154,Z 376.877,A -85,B 0,C 180,E1 -9639.515,E2 -9639.515} C_VEL
LIN {X 0,Y 425.691,Z 368.952,A -85,B 0,C 180,E1 -9640.945,E2 -9640.945} C_VEL
LIN {X 0,Y 426.418,Z 359.097,A -85,B 0,C 180,E1 -9642.372,E2 -9642.372} C_VEL
LIN {X 0,Y 427.175,Z 348.621,A -85,B 0,C 180,E1 -9643.573,E2 -9643.573} C_VEL
LIN {X 0,Y 427.716,Z 338.524,A -85,B 0,C 180,E1 -9644.512,E2 -9644.512} C_VEL
LIN {X 0,Y 428.462,Z 327.326,A -85,B 0,C 180,E1 -9645.337,E2 -9645.337} C_VEL
LIN {X 0,Y 429.03,Z 315.971,A -85,B 0,C 180,E1 -9645.986,E2 -9645.986} C_VEL
LIN {X 0,Y 429.553,Z 303.03,A -85,B 0,C 180,E1 -9646.516,E2 -9646.516} C_VEL
LIN {X 0,Y 429.875,Z 289.202,A -85,B 0,C 180,E1 -9646.87,E2 -9646.87} C_VEL
LIN {X 0,Y 430.61,Z 207.66,A -85,B 0,C 180,E1 -9648.24,E2 -9648.24} C_VEL
LIN {X 0,Y 426.854,Z 187.204,A -85,B 0,C 180,E1 -9648.784,E2 -9648.784} C_VEL
LIN {X 0,Y 426.829,Z 186.508,A -85,B 0,C 180,E1 -9648.859,E2 -9648.859} C_VEL
LIN {X 0,Y 427.611,Z 173.214,A -85,B 0,C 180,E1 -9651.703,E2 -9651.703} C_VEL
LIN {X 0,Y 425.81,Z 162.915,A -85,B 0,C 180,E1 -9654.11,E2 -9654.11} C_VEL
LIN {X 0,Y 425.32,Z 160.537,A -85,B 0,C 180,E1 -9654.751,E2 -9654.751} C_VEL
LIN {X 0,Y 425.35,Z 160.503,A -85,B 0,C 180,E1 -9657.557,E2 -9657.557} C_VEL
LIN {X 0,Y 425.289,Z 160.502,A -85,B 0,C 180,E1 -9660.816,E2 -9660.816} C_VEL
LIN {X 0,Y 425.312,Z 160.499,A -85,B 0,C 180,E1 -9664.288,E2 -9664.288} C_VEL
LIN {X 0,Y 425.278,Z 160.51,A -85,B 0,C 180,E1 -9667.694,E2 -9667.694} C_VEL
LIN {X 0,Y 425.278,Z 160.498,A -85,B 0,C 180,E1 -9670.52,E2 -9670.52} C_VEL
LIN {X 0,Y 425.255,Z 160.511,A -85,B 0,C 180,E1 -9673.35,E2 -9673.35} C_VEL
LIN {X 0,Y 425.254,Z 160.494,A -85,B 0,C 180,E1 -9676.649,E2 -9676.649} C_VEL
LIN {X 0,Y 425.292,Z 160.508,A -85,B 0,C 180,E1 -9679.873,E2 -9679.873} C_VEL
LIN {X 0,Y 425.275,Z 160.501,A -85,B 0,C 180,E1 -9682.488,E2 -9682.488} C_VEL
LIN {X 0,Y 425.304,Z 160.482,A -85,B 0,C 180,E1 -9685.817,E2 -9685.817} C_VEL
LIN {X 0,Y 425.286,Z 160.506,A -85,B 0,C 180,E1 -9689.238,E2 -9689.238} C_VEL
LIN {X 0,Y 425.344,Z 160.495,A -85,B 0,C 180,E1 -9692.442,E2 -9692.442} C_VEL
LIN {X 0,Y 425.342,Z 160.504,A -85,B 0,C 180,E1 -9695.601,E2 -9695.601} C_VEL
LIN {X 0,Y 425.287,Z 160.501,A -85,B 0,C 180,E1 -9698.681,E2 -9698.681} C_VEL
LIN {X 0,Y 425.327,Z 160.507,A -85,B 0,C 180,E1 -9701.702,E2 -9701.702} C_VEL
LIN {X 0,Y 425.341,Z 160.49,A -85,B 0,C 180,E1 -9704.67,E2 -9704.67} C_VEL
LIN {X 0,Y 425.406,Z 160.496,A -85,B 0,C 180,E1 -9707.598,E2 -9707.598} C_VEL
LIN {X 0,Y 425.436,Z 160.48,A -85,B 0,C 180,E1 -9711.45,E2 -9711.45} C_VEL
LIN {X 0,Y 425.542,Z 160.474,A -85,B 0,C 180,E1 -9714.313,E2 -9714.313} C_VEL
LIN {X 0,Y 425.564,Z 160.466,A -85,B 0,C 180,E1 -9718.107,E2 -9718.107} C_VEL
LIN {X 0,Y 425.693,Z 160.457,A -85,B 0,C 180,E1 -9720,E2 -9720} C_VEL
LIN {X 0,Y 425.537,Z 160.474,A -85,B 0,C 180,E1 -9722.84,E2 -9722.84} C_VEL
LIN {X 0,Y 425.539,Z 160.474,A -85,B 0,C 180,E1 -9725.687,E2 -9725.687} C_VEL
LIN {X 0,Y 425.401,Z 160.492,A -85,B 0,C 180,E1 -9728.551,E2 -9728.551} C_VEL
LIN {X 0,Y 425.405,Z 160.485,A -85,B 0,C 180,E1 -9732.402,E2 -9732.402} C_VEL
LIN {X 0,Y 425.381,Z 160.492,A -85,B 0,C 180,E1 -9736.312,E2 -9736.312} C_VEL
LIN {X 0,Y 425.322,Z 160.504,A -85,B 0,C 180,E1 -9739.636,E2 -9739.636} C_VEL
LIN {X 0,Y 425.282,Z 160.505,A -85,B 0,C 180,E1 -9742.339,E2 -9742.339} C_VEL
LIN {X 0,Y 425.286,Z 160.511,A -85,B 0,C 180,E1 -9745.446,E2 -9745.446} C_VEL
LIN {X 0,Y 425.343,Z 160.5,A -85,B 0,C 180,E1 -9747.558,E2 -9747.558} C_VEL
LIN {X 0,Y 425.283,Z 160.507,A -85,B 0,C 180,E1 -9750.817,E2 -9750.817} C_VEL
LIN {X 0,Y 425.305,Z 160.499,A -85,B 0,C 180,E1 -9754.288,E2 -9754.288} C_VEL
LIN {X 0,Y 425.274,Z 160.497,A -85,B 0,C 180,E1 -9757.695,E2 -9757.695} C_VEL
LIN {X 0,Y 425.273,Z 160.51,A -85,B 0,C 180,E1 -9760.52,E2 -9760.52} C_VEL
LIN {X 0,Y 425.258,Z 160.508,A -85,B 0,C 180,E1 -9763.957,E2 -9763.957} C_VEL
LIN {X 0,Y 425.247,Z 160.513,A -85,B 0,C 180,E1 -9766.651,E2 -9766.651} C_VEL
LIN {X 0,Y 425.259,Z 160.508,A -85,B 0,C 180,E1 -9769.87,E2 -9769.87} C_VEL
LIN {X 0,Y 425.274,Z 160.5,A -85,B 0,C 180,E1 -9772.489,E2 -9772.489} C_VEL
LIN {X 0,Y 425.306,Z 160.498,A -85,B 0,C 180,E1 -9775.818,E2 -9775.818} C_VEL
LIN {X 0,Y 425.29,Z 160.503,A -85,B 0,C 180,E1 -9779.239,E2 -9779.239} C_VEL
LIN {X 0,Y 425.27,Z 160.493,A -85,B 0,C 180,E1 -9782.437,E2 -9782.437} C_VEL
LIN {X 0,Y 425.318,Z 160.586,A -85,B 0,C 180,E1 -9783.965,E2 -9783.965} C_VEL
LIN {X 0,Y 427.443,Z 171.414,A -85,B 0,C 180,E1 -9786.502,E2 -9786.502} C_VEL
LIN {X 0,Y 427.911,Z 175.203,A -85,B 0,C 180,E1 -9787.341,E2 -9787.341} C_VEL
LIN {X 0,Y 426.792,Z 192.98,A -85,B 0,C 180,E1 -9791.046,E2 -9791.046} C_VEL
LIN {X 0,Y 426.799,Z 194.466,A -85,B 0,C 180,E1 -9791.258,E2 -9791.258} C_VEL
LIN {X 0,Y 430.599,Z 216.948,A -85,B 0,C 180,E1 -9791.835,E2 -9791.835} C_VEL
LIN {X 0,Y 429.768,Z 301.832,A -85,B 0,C 180,E1 -9793.279,E2 -9793.279} C_VEL
LIN {X 0,Y 429.238,Z 315.066,A -85,B 0,C 180,E1 -9793.686,E2 -9793.686} C_VEL
LIN {X 0,Y 428.725,Z 327.203,A -85,B 0,C 180,E1 -9794.246,E2 -9794.246} C_VEL
LIN {X 0,Y 428.03,Z 339.445,A -85,B 0,C 180,E1 -9795.013,E2 -9795.013} C_VEL
LIN {X 0,Y 427.361,Z 350.262,A -85,B 0,C 180,E1 -9795.891,E2 -9795.891} C_VEL
LIN {X 0,Y 426.654,Z 361.436,A -85,B 0,C 180,E1 -9797.03,E2 -9797.03} C_VEL
LIN {X 0,Y 426.018,Z 369.95,A -85,B 0,C 180,E1 -9798.099,E2 -9798.099} C_VEL
LIN {X 0,Y 425.454,Z 377.804,A -85,B 0,C 180,E1 -9799.29,E2 -9799.29} C_VEL
LIN {X 0,Y 424.915,Z 385.472,A -85,B 0,C 180,E1 -9800.72,E2 -9800.72} C_VEL
LIN {X 0,Y 424.505,Z 392.541,A -85,B 0,C 180,E1 -9802.389,E2 -9802.389} C_VEL
LIN {X 0,Y 424.255,Z 397.704,A -85,B 0,C 180,E1 -9803.975,E2 -9803.975} C_VEL
LIN {X 0,Y 424.213,Z 400.833,A -85,B 0,C 180,E1 -9805.248,E2 -9805.248} C_VEL
LIN {X 0,Y 424.1,Z 402.685,A -85,B 0,C 180,E1 -9806.199,E2 -9806.199} C_VEL
LIN {X 0,Y 424.122,Z 405.064,A -85,B 0,C 180,E1 -9808.1,E2 -9808.1} C_VEL
LIN {X 0,Y 424.062,Z 405.883,A -85,B 0,C 180,E1 -9810,E2 -9810} C_VEL
LIN {X 0,Y 424.122,Z 405.062,A -85,B 0,C 180,E1 -9811.899,E2 -9811.899} C_VEL
LIN {X 0,Y 424.094,Z 404.071,A -85,B 0,C 180,E1 -9812.849,E2 -9812.849} C_VEL
LIN {X 0,Y 424.1,Z 402.681,A -85,B 0,C 180,E1 -9813.8,E2 -9813.8} C_VEL
LIN {X 0,Y 424.25,Z 399.759,A -85,B 0,C 180,E1 -9815.227,E2 -9815.227} C_VEL
LIN {X 0,Y 424.387,Z 395.801,A -85,B 0,C 180,E1 -9816.656,E2 -9816.656} C_VEL
LIN {X 0,Y 424.655,Z 389.713,A -85,B 0,C 180,E1 -9818.326,E2 -9818.326} C_VEL
LIN {X 0,Y 425.066,Z 383.059,A -85,B 0,C 180,E1 -9819.756,E2 -9819.756} C_VEL
LIN {X 0,Y 425.622,Z 374.801,A -85,B 0,C 180,E1 -9821.187,E2 -9821.187} C_VEL
LIN {X 0,Y 426.282,Z 366.335,A -85,B 0,C 180,E1 -9822.375,E2 -9822.375} C_VEL
LIN {X 0,Y 426.984,Z 356.584,A -85,B 0,C 180,E1 -9823.491,E2 -9823.491} C_VEL
LIN {X 0,Y 427.623,Z 345.511,A -85,B 0,C 180,E1 -9824.514,E2 -9824.514} C_VEL
LIN {X 0,Y 428.288,Z 334.151,A -85,B 0,C 180,E1 -9825.343,E2 -9825.343} C_VEL
LIN {X 0,Y 428.926,Z 322.489,A -85,B 0,C 180,E1 -9825.989,E2 -9825.989} C_VEL
LIN {X 0,Y 429.474,Z 309.042,A -85,B 0,C 180,E1 -9826.518,E2 -9826.518} C_VEL
LIN {X 0,Y 429.817,Z 295.721,A -85,B 0,C 180,E1 -9826.84,E2 -9826.84} C_VEL
LIN {X 0,Y 430.561,Z 216.141,A -85,B 0,C 180,E1 -9828.173,E2 -9828.173} C_VEL
LIN {X 0,Y 426.791,Z 194.312,A -85,B 0,C 180,E1 -9828.74,E2 -9828.74} C_VEL
LIN {X 0,Y 426.926,Z 190.45,A -85,B 0,C 180,E1 -9829.471,E2 -9829.471} C_VEL
LIN {X 0,Y 427.892,Z 175.19,A -85,B 0,C 180,E1 -9832.655,E2 -9832.655} C_VEL
LIN {X 0,Y 427.016,Z 168.988,A -85,B 0,C 180,E1 -9834.037,E2 -9834.037} C_VEL
LIN {X 0,Y 425.313,Z 160.574,A -85,B 0,C 180,E1 -9836.034,E2 -9836.034} C_VEL
LIN {X 0,Y 425.31,Z 160.505,A -85,B 0,C 180,E1 -9838.861,E2 -9838.861} C_VEL
LIN {X 0,Y 425.261,Z 160.513,A -85,B 0,C 180,E1 -9841.926,E2 -9841.926} C_VEL
LIN {X 0,Y 425.294,Z 160.51,A -85,B 0,C 180,E1 -9845.335,E2 -9845.335} C_VEL
LIN {X 0,Y 425.276,Z 160.497,A -85,B 0,C 180,E1 -9848.899,E2 -9848.899} C_VEL
LIN {X 0,Y 425.276,Z 160.507,A -85,B 0,C 180,E1 -9851.956,E2 -9851.956} C_VEL
LIN {X 0,Y 425.278,Z 160.51,A -85,B 0,C 180,E1 -9855.282,E2 -9855.282} C_VEL
LIN {X 0,Y 425.267,Z 160.51,A -85,B 0,C 180,E1 -9858.62,E2 -9858.62} C_VEL
LIN {X 0,Y 425.29,Z 160.5,A -85,B 0,C 180,E1 -9861.1,E2 -9861.1} C_VEL
LIN {X 0,Y 425.29,Z 160.49,A -85,B 0,C 180,E1 -9864.663,E2 -9864.663} C_VEL
LIN {X 0,Y 425.254,Z 160.511,A -85,B 0,C 180,E1 -9868.072,E2 -9868.072} C_VEL
LIN {X 0,Y 425.32,Z 160.502,A -85,B 0,C 180,E1 -9871.367,E2 -9871.367} C_VEL
LIN {X 0,Y 425.343,Z 160.5,A -85,B 0,C 180,E1 -9873.505,E2 -9873.505} C_VEL
LIN {X 0,Y 425.273,Z 160.504,A -85,B 0,C 180,E1 -9876.633,E2 -9876.633} C_VEL
LIN {X 0,Y 425.283,Z 160.506,A -85,B 0,C 180,E1 -9879.694,E2 -9879.694} C_VEL
LIN {X 0,Y 425.321,Z 160.498,A -85,B 0,C 180,E1 -9882.697,E2 -9882.697} C_VEL
LIN {X 0,Y 425.341,Z 160.499,A -85,B 0,C 180,E1 -9885.65,E2 -9885.65} C_VEL
LIN {X 0,Y 425.358,Z 160.492,A -85,B 0,C 180,E1 -9888.564,E2 -9888.564} C_VEL
LIN {X 0,Y 425.526,Z 160.481,A -85,B 0,C 180,E1 -9892.407,E2 -9892.407} C_VEL
LIN {X 0,Y 425.536,Z 160.474,A -85,B 0,C 180,E1 -9894.313,E2 -9894.313} C_VEL
LIN {X 0,Y 425.561,Z 160.473,A -85,B 0,C 180,E1 -9898.107,E2 -9898.107} C_VEL
LIN {X 0,Y 425.689,Z 160.457,A -85,B 0,C 180,E1 -9900,E2 -9900} C_VEL
LIN {X 0,Y 425.532,Z 160.471,A -85,B 0,C 180,E1 -9902.84,E2 -9902.84} C_VEL
LIN {X 0,Y 425.514,Z 160.479,A -85,B 0,C 180,E1 -9906.639,E2 -9906.639} C_VEL
LIN {X 0,Y 425.389,Z 160.482,A -85,B 0,C 180,E1 -9909.51,E2 -9909.51} C_VEL
LIN {X 0,Y 425.382,Z 160.494,A -85,B 0,C 180,E1 -9912.904,E2 -9912.904} C_VEL
LIN {X 0,Y 425.35,Z 160.497,A -85,B 0,C 180,E1 -9916.605,E2 -9916.605} C_VEL
LIN {X 0,Y 425.318,Z 160.503,A -85,B 0,C 180,E1 -9919.636,E2 -9919.636} C_VEL
LIN {X 0,Y 425.297,Z 160.501,A -85,B 0,C 180,E1 -9923.366,E2 -9923.366} C_VEL
LIN {X 0,Y 425.337,Z 160.495,A -85,B 0,C 180,E1 -9926.845,E2 -9926.845} C_VEL
LIN {X 0,Y 425.281,Z 160.508,A -85,B 0,C 180,E1 -9929.72,E2 -9929.72} C_VEL
LIN {X 0,Y 425.273,Z 160.499,A -85,B 0,C 180,E1 -9933.049,E2 -9933.049} C_VEL
LIN {X 0,Y 425.274,Z 160.486,A -85,B 0,C 180,E1 -9935.93,E2 -9935.93} C_VEL
LIN {X 0,Y 425.286,Z 160.506,A -85,B 0,C 180,E1 -9939.044,E2 -9939.044} C_VEL
LIN {X 0,Y 425.268,Z 160.494,A -85,B 0,C 180,E1 -9942.654,E2 -9942.654} C_VEL
LIN {X 0,Y 425.256,Z 160.514,A -85,B 0,C 180,E1 -9946.045,E2 -9946.045} C_VEL
LIN {X 0,Y 425.268,Z 160.503,A -85,B 0,C 180,E1 -9948.622,E2 -9948.622} C_VEL
LIN {X 0,Y 425.292,Z 160.498,A -85,B 0,C 180,E1 -9951.102,E2 -9951.102} C_VEL
LIN {X 0,Y 425.297,Z 160.498,A -85,B 0,C 180,E1 -9954.665,E2 -9954.665} C_VEL
LIN {X 0,Y 425.262,Z 160.508,A -85,B 0,C 180,E1 -9958.074,E2 -9958.074} C_VEL
LIN {X 0,Y 425.329,Z 160.502,A -85,B 0,C 180,E1 -9961.369,E2 -9961.369} C_VEL
LIN {X 0,Y 425.293,Z 160.511,A -85,B 0,C 180,E1 -9964.556,E2 -9964.556} C_VEL
LIN {X 0,Y 425.375,Z 160.734,A -85,B 0,C 180,E1 -9965.444,E2 -9965.444} C_VEL
LIN {X 0,Y 427.452,Z 171.63,A -85,B 0,C 180,E1 -9968.036,E2 -9968.036} C_VEL
LIN {X 0,Y 427.393,Z 176.218,A -85,B 0,C 180,E1 -9969.045,E2 -9969.045} C_VEL
LIN {X 0,Y 426.826,Z 186.761,A -85,B 0,C 180,E1 -9971.275,E2 -9971.275} C_VEL
LIN {X 0,Y 427.361,Z 190.061,A -85,B 0,C 180,E1 -9971.407,E2 -9971.407} C_VEL
LIN {X 0,Y 430.642,Z 208.488,A -85,B 0,C 180,E1 -9971.872,E2 -9971.872} C_VEL
LIN {X 0,Y 429.79,Z 294.695,A -85,B 0,C 180,E1 -9973.342,E2 -9973.342} C_VEL
LIN {X 0,Y 429.395,Z 307.021,A -85,B 0,C 180,E1 -9973.723,E2 -9973.723} C_VEL
LIN {X 0,Y 428.776,Z 319.841,A -85,B 0,C 180,E1 -9974.31,E2 -9974.31} C_VEL
LIN {X 0,Y 428.154,Z 331.326,A -85,B 0,C 180,E1 -9975.026,E2 -9975.026} C_VEL
LIN {X 0,Y 427.556,Z 342.042,A -85,B 0,C 180,E1 -9975.888,E2 -9975.888} C_VEL
LIN {X 0,Y 426.922,Z 352.318,A -85,B 0,C 180,E1 -9976.918,E2 -9976.918} C_VEL
LIN {X 0,Y 426.668,Z 356.456,A -85,B 0,C 180,E1 -9977.4,E2 -9977.4} C_VEL
LIN {X 0,Y 425.609,Z 360.799,A -85,B 0,C 180,E1 -9977.928,E2 -9977.928} C_VEL
LIN {X 0,Y 422.22,Z 367.46,A -85,B 0,C 180,E1 -9978.811,E2 -9978.811} C_VEL
LIN {X 0,Y 418.969,Z 373.568,A -85,B 0,C 180,E1 -9979.776,E2 -9979.776} C_VEL
LIN {X 0,Y 418.129,Z 376.948,A -85,B 0,C 180,E1 -9980.425,E2 -9980.425} C_VEL
LIN {X 0,Y 417.694,Z 382.905,A -85,B 0,C 180,E1 -9981.778,E2 -9981.778} C_VEL
LIN {X 0,Y 417.394,Z 388.605,A -85,B 0,C 180,E1 -9983.431,E2 -9983.431} C_VEL
LIN {X 0,Y 417.187,Z 393.058,A -85,B 0,C 180,E1 -9985.169,E2 -9985.169} C_VEL
LIN {X 0,Y 417.064,Z 394.927,A -85,B 0,C 180,E1 -9986.136,E2 -9986.136} C_VEL
LIN {X 0,Y 417.052,Z 396.335,A -85,B 0,C 180,E1 -9987.103,E2 -9987.103} C_VEL
LIN {X 0,Y 417.059,Z 397.336,A -85,B 0,C 180,E1 -9988.069,E2 -9988.069} C_VEL
LIN {X 0,Y 416.983,Z 398.188,A -85,B 0,C 180,E1 -9990,E2 -9990} C_VEL
LIN {X 0,Y 416.994,Z 398,A -85,B 0,C 180,E1 -9990.966,E2 -9990.966} C_VEL
LIN {X 0,Y 417.06,Z 397.412,A -85,B 0,C 180,E1 -9991.932,E2 -9991.932} C_VEL
LIN {X 0,Y 417.061,Z 395.081,A -85,B 0,C 180,E1 -9993.865,E2 -9993.865} C_VEL
LIN {X 0,Y 417.241,Z 392.203,A -85,B 0,C 180,E1 -9995.316,E2 -9995.316} C_VEL
LIN {X 0,Y 417.421,Z 388.302,A -85,B 0,C 180,E1 -9996.769,E2 -9996.769} C_VEL
LIN {X 0,Y 417.659,Z 383.271,A -85,B 0,C 180,E1 -9998.223,E2 -9998.223} C_VEL
LIN {X 0,Y 418.126,Z 376.94,A -85,B 0,C 180,E1 -9999.677,E2 -9999.677} C_VEL
LIN {X 0,Y 418.69,Z 369.015,A -85,B 0,C 180,E1 -10001.13,E2 -10001.13} C_VEL
LIN {X 0,Y 419.482,Z 359.159,A -85,B 0,C 180,E1 -10002.58,E2 -10002.58} C_VEL
LIN {X 0,Y 420.215,Z 349.431,A -85,B 0,C 180,E1 -10003.724,E2 -10003.724} C_VEL
LIN {X 0,Y 420.853,Z 338.583,A -85,B 0,C 180,E1 -10004.754,E2 -10004.754} C_VEL
LIN {X 0,Y 421.626,Z 327.384,A -85,B 0,C 180,E1 -10005.592,E2 -10005.592} C_VEL
LIN {X 0,Y 422.217,Z 316.028,A -85,B 0,C 180,E1 -10006.251,E2 -10006.251} C_VEL
LIN {X 0,Y 422.763,Z 303.082,A -85,B 0,C 180,E1 -10006.789,E2 -10006.789} C_VEL
LIN {X 0,Y 423.102,Z 289.245,A -85,B 0,C 180,E1 -10007.148,E2 -10007.148} C_VEL
LIN {X 0,Y 423.761,Z 207.543,A -85,B 0,C 180,E1 -10008.548,E2 -10008.548} C_VEL
LIN {X 0,Y 419.931,Z 187.074,A -85,B 0,C 180,E1 -10009.115,E2 -10009.115} C_VEL
